LIN {X 0,Y 573.313,Z 246.817,A -85,B 0,C 180,E1 -2273.642,E2 -2273.642} C_VEL
LIN {X 0,Y 573.236,Z 246.702,A -85,B 0,C 180,E1 -2276.492,E2 -2276.492} C_VEL
LIN {X 0,Y 573.238,Z 246.706,A -85,B 0,C 180,E1 -2278.564,E2 -2278.564} C_VEL
LIN {X 0,Y 573.228,Z 246.705,A -85,B 0,C 180,E1 -2280.992,E2 -2280.992} C_VEL
LIN {X 0,Y 573.26,Z 246.695,A -85,B 0,C 180,E1 -2283.523,E2 -2283.523} C_VEL
LIN {X 0,Y 573.212,Z 246.707,A -85,B 0,C 180,E1 -2286.051,E2 -2286.051} C_VEL
LIN {X 0,Y 573.239,Z 246.706,A -85,B 0,C 180,E1 -2288.701,E2 -2288.701} C_VEL
LIN {X 0,Y 573.25,Z 246.695,A -85,B 0,C 180,E1 -2291.595,E2 -2291.595} C_VEL
LIN {X 0,Y 573.235,Z 246.71,A -85,B 0,C 180,E1 -2294.332,E2 -2294.332} C_VEL
LIN {X 0,Y 573.235,Z 246.7,A -85,B 0,C 180,E1 -2297.358,E2 -2297.358} C_VEL
LIN {X 0,Y 573.244,Z 246.706,A -85,B 0,C 180,E1 -2300.393,E2 -2300.393} C_VEL
LIN {X 0,Y 573.251,Z 246.697,A -85,B 0,C 180,E1 -2303.077,E2 -2303.077} C_VEL
LIN {X 0,Y 573.268,Z 246.693,A -85,B 0,C 180,E1 -2305.671,E2 -2305.671} C_VEL
LIN {X 0,Y 573.242,Z 246.707,A -85,B 0,C 180,E1 -2308.185,E2 -2308.185} C_VEL
LIN {X 0,Y 573.262,Z 246.698,A -85,B 0,C 180,E1 -2310.634,E2 -2310.634} C_VEL
LIN {X 0,Y 573.264,Z 246.698,A -85,B 0,C 180,E1 -2313.5,E2 -2313.5} C_VEL
LIN {X 0,Y 573.227,Z 246.707,A -85,B 0,C 180,E1 -2316.134,E2 -2316.134} C_VEL
LIN {X 0,Y 573.243,Z 246.699,A -85,B 0,C 180,E1 -2319.173,E2 -2319.173} C_VEL
LIN {X 0,Y 573.23,Z 246.704,A -85,B 0,C 180,E1 -2321.412,E2 -2321.412} C_VEL
LIN {X 0,Y 573.252,Z 246.703,A -85,B 0,C 180,E1 -2323.622,E2 -2323.622} C_VEL
LIN {X 0,Y 573.231,Z 246.701,A -85,B 0,C 180,E1 -2326.529,E2 -2326.529} C_VEL
LIN {X 0,Y 573.253,Z 246.696,A -85,B 0,C 180,E1 -2328.745,E2 -2328.745} C_VEL
LIN {X 0,Y 573.283,Z 246.701,A -85,B 0,C 180,E1 -2331.541,E2 -2331.541} C_VEL
LIN {X 0,Y 573.286,Z 246.693,A -85,B 0,C 180,E1 -2334.372,E2 -2334.372} C_VEL
LIN {X 0,Y 573.301,Z 246.696,A -85,B 0,C 180,E1 -2337.892,E2 -2337.892} C_VEL
LIN {X 0,Y 573.328,Z 246.688,A -85,B 0,C 180,E1 -2340.702,E2 -2340.702} C_VEL
LIN {X 0,Y 573.233,Z 246.709,A -85,B 0,C 180,E1 -2343.515,E2 -2343.515} C_VEL
LIN {X 0,Y 573.286,Z 246.7,A -85,B 0,C 180,E1 -2345.628,E2 -2345.628} C_VEL
LIN {X 0,Y 573.283,Z 246.692,A -85,B 0,C 180,E1 -2348.46,E2 -2348.46} C_VEL
LIN {X 0,Y 573.262,Z 246.706,A -85,B 0,C 180,E1 -2351.312,E2 -2351.312} C_VEL
LIN {X 0,Y 573.265,Z 246.695,A -85,B 0,C 180,E1 -2354.193,E2 -2354.193} C_VEL
LIN {X 0,Y 573.252,Z 246.706,A -85,B 0,C 180,E1 -2357.112,E2 -2357.112} C_VEL
LIN {X 0,Y 573.247,Z 246.697,A -85,B 0,C 180,E1 -2360.077,E2 -2360.077} C_VEL
LIN {X 0,Y 573.226,Z 246.711,A -85,B 0,C 180,E1 -2363.1,E2 -2363.1} C_VEL
LIN {X 0,Y 573.244,Z 246.7,A -85,B 0,C 180,E1 -2364.396,E2 -2364.396} C_VEL
LIN {X 0,Y 572.617,Z 246.786,A -85,B 0,C 180,E1 -2364.983,E2 -2364.983} C_VEL
LIN {X 0,Y 569.776,Z 247.14,A -85,B 0,C 180,E1 -2365.934,E2 -2365.934} C_VEL
LIN {X 0,Y 567.346,Z 247.442,A -85,B 0,C 180,E1 -2366.7,E2 -2366.7} C_VEL
LIN {X 0,Y 566.295,Z 247.57,A -85,B 0,C 180,E1 -2367.291,E2 -2367.291} C_VEL
LIN {X 0,Y 566.207,Z 247.578,A -85,B 0,C 180,E1 -2367.491,E2 -2367.491} C_VEL
LIN {X 0,Y 566.22,Z 247.574,A -85,B 0,C 180,E1 -2369.768,E2 -2369.768} C_VEL
LIN {X 0,Y 566.201,Z 247.575,A -85,B 0,C 180,E1 -2372.431,E2 -2372.431} C_VEL
LIN {X 0,Y 566.209,Z 247.582,A -85,B 0,C 180,E1 -2374.995,E2 -2374.995} C_VEL
LIN {X 0,Y 566.192,Z 247.579,A -85,B 0,C 180,E1 -2377.461,E2 -2377.461} C_VEL
LIN {X 0,Y 566.222,Z 247.574,A -85,B 0,C 180,E1 -2380.198,E2 -2380.198} C_VEL
LIN {X 0,Y 566.197,Z 247.581,A -85,B 0,C 180,E1 -2383.055,E2 -2383.055} C_VEL
LIN {X 0,Y 566.199,Z 247.578,A -85,B 0,C 180,E1 -2386.049,E2 -2386.049} C_VEL
LIN {X 0,Y 566.209,Z 247.581,A -85,B 0,C 180,E1 -2388.865,E2 -2388.865} C_VEL
LIN {X 0,Y 566.184,Z 247.577,A -85,B 0,C 180,E1 -2391.638,E2 -2391.638} C_VEL
LIN {X 0,Y 566.195,Z 247.584,A -85,B 0,C 180,E1 -2394.311,E2 -2394.311} C_VEL
LIN {X 0,Y 566.228,Z 247.577,A -85,B 0,C 180,E1 -2396.899,E2 -2396.899} C_VEL
LIN {X 0,Y 566.18,Z 247.58,A -85,B 0,C 180,E1 -2399.408,E2 -2399.408} C_VEL
LIN {X 0,Y 566.212,Z 247.575,A -85,B 0,C 180,E1 -2401.858,E2 -2401.858} C_VEL
LIN {X 0,Y 566.216,Z 247.582,A -85,B 0,C 180,E1 -2404.252,E2 -2404.252} C_VEL
LIN {X 0,Y 566.24,Z 247.699,A -85,B 0,C 180,E1 -2407.28,E2 -2407.28} C_VEL
LIN {X 0,Y 567.062,Z 253.165,A -85,B 0,C 180,E1 -2408.173,E2 -2408.173} C_VEL
LIN {X 0,Y 566.746,Z 272.236,A -85,B 0,C 180,E1 -2411.01,E2 -2411.01} C_VEL
LIN {X 0,Y 566.631,Z 286.377,A -85,B 0,C 180,E1 -2413.053,E2 -2413.053} C_VEL
LIN {X 0,Y 567.533,Z 291.478,A -85,B 0,C 180,E1 -2413.174,E2 -2413.174} C_VEL
LIN {X 0,Y 567.785,Z 300.796,A -85,B 0,C 180,E1 -2413.302,E2 -2413.302} C_VEL
LIN {X 0,Y 567.442,Z 423.944,A -85,B 0,C 180,E1 -2414.902,E2 -2414.902} C_VEL
LIN {X 0,Y 567.321,Z 438.302,A -85,B 0,C 180,E1 -2415.239,E2 -2415.239} C_VEL
LIN {X 0,Y 567.131,Z 452.855,A -85,B 0,C 180,E1 -2415.742,E2 -2415.742} C_VEL
LIN {X 0,Y 566.944,Z 466.542,A -85,B 0,C 180,E1 -2416.377,E2 -2416.377} C_VEL
LIN {X 0,Y 566.744,Z 478.824,A -85,B 0,C 180,E1 -2417.103,E2 -2417.103} C_VEL
LIN {X 0,Y 566.56,Z 491.218,A -85,B 0,C 180,E1 -2418.008,E2 -2418.008} C_VEL
LIN {X 0,Y 566.434,Z 502.054,A -85,B 0,C 180,E1 -2418.98,E2 -2418.98} C_VEL
LIN {X 0,Y 566.215,Z 511.482,A -85,B 0,C 180,E1 -2419.993,E2 -2419.993} C_VEL
LIN {X 0,Y 566.133,Z 519.865,A -85,B 0,C 180,E1 -2421.073,E2 -2421.073} C_VEL
LIN {X 0,Y 566.047,Z 527.875,A -85,B 0,C 180,E1 -2422.33,E2 -2422.33} C_VEL
LIN {X 0,Y 565.945,Z 534.324,A -85,B 0,C 180,E1 -2423.583,E2 -2423.583} C_VEL
LIN {X 0,Y 565.928,Z 538.8,A -85,B 0,C 180,E1 -2424.656,E2 -2424.656} C_VEL
LIN {X 0,Y 565.957,Z 542.312,A -85,B 0,C 180,E1 -2425.727,E2 -2425.727} C_VEL
LIN {X 0,Y 565.875,Z 545.744,A -85,B 0,C 180,E1 -2427.152,E2 -2427.152} C_VEL
LIN {X 0,Y 565.844,Z 547.785,A -85,B 0,C 180,E1 -2428.577,E2 -2428.577} C_VEL
LIN {X 0,Y 565.838,Z 548.496,A -85,B 0,C 180,E1 -2430,E2 -2430} C_VEL
LIN {X 0,Y 565.841,Z 547.88,A -85,B 0,C 180,E1 -2431.423,E2 -2431.423} C_VEL
LIN {X 0,Y 565.873,Z 545.923,A -85,B 0,C 180,E1 -2432.847,E2 -2432.847} C_VEL
LIN {X 0,Y 565.958,Z 542.577,A -85,B 0,C 180,E1 -2434.273,E2 -2434.273} C_VEL
LIN {X 0,Y 565.983,Z 537.749,A -85,B 0,C 180,E1 -2435.701,E2 -2435.701} C_VEL
LIN {X 0,Y 565.981,Z 531.282,A -85,B 0,C 180,E1 -2437.133,E2 -2437.133} C_VEL
LIN {X 0,Y 566.093,Z 524.083,A -85,B 0,C 180,E1 -2438.388,E2 -2438.388} C_VEL
LIN {X 0,Y 566.172,Z 516.544,A -85,B 0,C 180,E1 -2439.466,E2 -2439.466} C_VEL
LIN {X 0,Y 566.29,Z 507.487,A -85,B 0,C 180,E1 -2440.548,E2 -2440.548} C_VEL
LIN {X 0,Y 566.47,Z 496.523,A -85,B 0,C 180,E1 -2441.631,E2 -2441.631} C_VEL
LIN {X 0,Y 566.631,Z 485.35,A -85,B 0,C 180,E1 -2442.536,E2 -2442.536} C_VEL
LIN {X 0,Y 566.843,Z 473,A -85,B 0,C 180,E1 -2443.351,E2 -2443.351} C_VEL
LIN {X 0,Y 567.064,Z 461.118,A -85,B 0,C 180,E1 -2443.985,E2 -2443.985} C_VEL
LIN {X 0,Y 567.234,Z 448.803,A -85,B 0,C 180,E1 -2444.507,E2 -2444.507} C_VEL
LIN {X 0,Y 567.352,Z 434.83,A -85,B 0,C 180,E1 -2444.947,E2 -2444.947} C_VEL
LIN {X 0,Y 567.451,Z 421.093,A -85,B 0,C 180,E1 -2445.236,E2 -2445.236} C_VEL
LIN {X 0,Y 567.731,Z 292.506,A -85,B 0,C 180,E1 -2446.897,E2 -2446.897} C_VEL
LIN {X 0,Y 566.636,Z 286.481,A -85,B 0,C 180,E1 -2447.029,E2 -2447.029} C_VEL
LIN {X 0,Y 566.788,Z 269.863,A -85,B 0,C 180,E1 -2449.429,E2 -2449.429} C_VEL
LIN {X 0,Y 567.066,Z 252.496,A -85,B 0,C 180,E1 -2452.018,E2 -2452.018} C_VEL
LIN {X 0,Y 566.246,Z 247.694,A -85,B 0,C 180,E1 -2452.812,E2 -2452.812} C_VEL
LIN {X 0,Y 566.215,Z 247.58,A -85,B 0,C 180,E1 -2455.748,E2 -2455.748} C_VEL
LIN {X 0,Y 566.202,Z 247.576,A -85,B 0,C 180,E1 -2458.201,E2 -2458.201} C_VEL
LIN {X 0,Y 566.189,Z 247.58,A -85,B 0,C 180,E1 -2461.076,E2 -2461.076} C_VEL
LIN {X 0,Y 566.21,Z 247.582,A -85,B 0,C 180,E1 -2463.733,E2 -2463.733} C_VEL
LIN {X 0,Y 566.208,Z 247.576,A -85,B 0,C 180,E1 -2466.568,E2 -2466.568} C_VEL
LIN {X 0,Y 566.207,Z 247.583,A -85,B 0,C 180,E1 -2469.684,E2 -2469.684} C_VEL
LIN {X 0,Y 566.211,Z 247.573,A -85,B 0,C 180,E1 -2472.086,E2 -2472.086} C_VEL
LIN {X 0,Y 566.169,Z 247.584,A -85,B 0,C 180,E1 -2475.035,E2 -2475.035} C_VEL
LIN {X 0,Y 566.207,Z 247.571,A -85,B 0,C 180,E1 -2478.136,E2 -2478.136} C_VEL
LIN {X 0,Y 566.217,Z 247.575,A -85,B 0,C 180,E1 -2480.726,E2 -2480.726} C_VEL
LIN {X 0,Y 566.212,Z 247.576,A -85,B 0,C 180,E1 -2483.783,E2 -2483.783} C_VEL
LIN {X 0,Y 566.206,Z 247.57,A -85,B 0,C 180,E1 -2486.265,E2 -2486.265} C_VEL
LIN {X 0,Y 566.196,Z 247.58,A -85,B 0,C 180,E1 -2488.921,E2 -2488.921} C_VEL
LIN {X 0,Y 566.189,Z 247.587,A -85,B 0,C 180,E1 -2491.046,E2 -2491.046} C_VEL
LIN {X 0,Y 566.208,Z 247.577,A -85,B 0,C 180,E1 -2493.458,E2 -2493.458} C_VEL
LIN {X 0,Y 566.192,Z 247.578,A -85,B 0,C 180,E1 -2495.819,E2 -2495.819} C_VEL
LIN {X 0,Y 566.2,Z 247.584,A -85,B 0,C 180,E1 -2498.902,E2 -2498.902} C_VEL
LIN {X 0,Y 566.204,Z 247.581,A -85,B 0,C 180,E1 -2501.172,E2 -2501.172} C_VEL
LIN {X 0,Y 566.213,Z 247.576,A -85,B 0,C 180,E1 -2503.412,E2 -2503.412} C_VEL
LIN {X 0,Y 566.194,Z 247.578,A -85,B 0,C 180,E1 -2506.359,E2 -2506.359} C_VEL
LIN {X 0,Y 566.266,Z 247.576,A -85,B 0,C 180,E1 -2508.654,E2 -2508.654} C_VEL
LIN {X 0,Y 566.226,Z 247.571,A -85,B 0,C 180,E1 -2511.434,E2 -2511.434} C_VEL
LIN {X 0,Y 566.254,Z 247.574,A -85,B 0,C 180,E1 -2514.302,E2 -2514.302} C_VEL
LIN {X 0,Y 566.271,Z 247.565,A -85,B 0,C 180,E1 -2517.866,E2 -2517.866} C_VEL
LIN {X 0,Y 566.299,Z 247.571,A -85,B 0,C 180,E1 -2520.711,E2 -2520.711} C_VEL
LIN {X 0,Y 566.27,Z 247.569,A -85,B 0,C 180,E1 -2522.846,E2 -2522.846} C_VEL
LIN {X 0,Y 566.253,Z 247.569,A -85,B 0,C 180,E1 -2525.698,E2 -2525.698} C_VEL
LIN {X 0,Y 566.24,Z 247.577,A -85,B 0,C 180,E1 -2528.565,E2 -2528.565} C_VEL
LIN {X 0,Y 566.232,Z 247.571,A -85,B 0,C 180,E1 -2531.454,E2 -2531.454} C_VEL
LIN {X 0,Y 566.225,Z 247.578,A -85,B 0,C 180,E1 -2534.507,E2 -2534.507} C_VEL
LIN {X 0,Y 566.195,Z 247.575,A -85,B 0,C 180,E1 -2537.332,E2 -2537.332} C_VEL
LIN {X 0,Y 566.206,Z 247.581,A -85,B 0,C 180,E1 -2540.337,E2 -2540.337} C_VEL
LIN {X 0,Y 566.182,Z 247.578,A -85,B 0,C 180,E1 -2543.404,E2 -2543.404} C_VEL
LIN {X 0,Y 566.207,Z 247.581,A -85,B 0,C 180,E1 -2545.749,E2 -2545.749} C_VEL
LIN {X 0,Y 566.198,Z 247.583,A -85,B 0,C 180,E1 -2548.203,E2 -2548.203} C_VEL
LIN {X 0,Y 566.186,Z 247.579,A -85,B 0,C 180,E1 -2550.592,E2 -2550.592} C_VEL
LIN {X 0,Y 566.221,Z 247.57,A -85,B 0,C 180,E1 -2553.102,E2 -2553.102} C_VEL
LIN {X 0,Y 566.206,Z 247.576,A -85,B 0,C 180,E1 -2555.689,E2 -2555.689} C_VEL
LIN {X 0,Y 566.21,Z 247.576,A -85,B 0,C 180,E1 -2558.56,E2 -2558.56} C_VEL
LIN {X 0,Y 566.206,Z 247.576,A -85,B 0,C 180,E1 -2561.137,E2 -2561.137} C_VEL
LIN {X 0,Y 566.192,Z 247.582,A -85,B 0,C 180,E1 -2564.036,E2 -2564.036} C_VEL
LIN {X 0,Y 566.205,Z 247.577,A -85,B 0,C 180,E1 -2567.083,E2 -2567.083} C_VEL
LIN {X 0,Y 566.223,Z 247.58,A -85,B 0,C 180,E1 -2569.803,E2 -2569.803} C_VEL
LIN {X 0,Y 566.195,Z 247.575,A -85,B 0,C 180,E1 -2572.6,E2 -2572.6} C_VEL
LIN {X 0,Y 566.201,Z 247.582,A -85,B 0,C 180,E1 -2575.183,E2 -2575.183} C_VEL
LIN {X 0,Y 566.233,Z 247.578,A -85,B 0,C 180,E1 -2577.744,E2 -2577.744} C_VEL
LIN {X 0,Y 566.202,Z 247.57,A -85,B 0,C 180,E1 -2580.329,E2 -2580.329} C_VEL
LIN {X 0,Y 566.21,Z 247.578,A -85,B 0,C 180,E1 -2582.662,E2 -2582.662} C_VEL
LIN {X 0,Y 566.236,Z 247.578,A -85,B 0,C 180,E1 -2585.04,E2 -2585.04} C_VEL
LIN {X 0,Y 566.263,Z 247.807,A -85,B 0,C 180,E1 -2586.212,E2 -2586.212} C_VEL
LIN {X 0,Y 567.195,Z 253.103,A -85,B 0,C 180,E1 -2587.027,E2 -2587.027} C_VEL
LIN {X 0,Y 566.934,Z 273.326,A -85,B 0,C 180,E1 -2589.88,E2 -2589.88} C_VEL
LIN {X 0,Y 566.604,Z 294.059,A -85,B 0,C 180,E1 -2592.763,E2 -2592.763} C_VEL
LIN {X 0,Y 566.662,Z 296.302,A -85,B 0,C 180,E1 -2593.024,E2 -2593.024} C_VEL
LIN {X 0,Y 567.795,Z 303.619,A -85,B 0,C 180,E1 -2593.165,E2 -2593.165} C_VEL
LIN {X 0,Y 567.456,Z 432.658,A -85,B 0,C 180,E1 -2594.833,E2 -2594.833} C_VEL
LIN {X 0,Y 567.301,Z 447.176,A -85,B 0,C 180,E1 -2595.16,E2 -2595.16} C_VEL
LIN {X 0,Y 567.19,Z 460.406,A -85,B 0,C 180,E1 -2595.599,E2 -2595.599} C_VEL
LIN {X 0,Y 567.011,Z 473.883,A -85,B 0,C 180,E1 -2596.196,E2 -2596.196} C_VEL
LIN {X 0,Y 566.77,Z 486.683,A -85,B 0,C 180,E1 -2596.921,E2 -2596.921} C_VEL
LIN {X 0,Y 566.615,Z 498.316,A -85,B 0,C 180,E1 -2597.737,E2 -2597.737} C_VEL
LIN {X 0,Y 566.443,Z 508.224,A -85,B 0,C 180,E1 -2598.572,E2 -2598.572} C_VEL
LIN {X 0,Y 566.294,Z 518.709,A -85,B 0,C 180,E1 -2599.633,E2 -2599.633} C_VEL
LIN {X 0,Y 566.18,Z 527.56,A -85,B 0,C 180,E1 -2600.714,E2 -2600.714} C_VEL
LIN {X 0,Y 566.047,Z 536.037,A -85,B 0,C 180,E1 -2601.971,E2 -2601.971} C_VEL
LIN {X 0,Y 565.966,Z 543.803,A -85,B 0,C 180,E1 -2603.422,E2 -2603.422} C_VEL
LIN {X 0,Y 565.928,Z 548.961,A -85,B 0,C 180,E1 -2604.656,E2 -2604.656} C_VEL
LIN {X 0,Y 565.956,Z 552.444,A -85,B 0,C 180,E1 -2605.727,E2 -2605.727} C_VEL
LIN {X 0,Y 565.875,Z 555.832,A -85,B 0,C 180,E1 -2607.153,E2 -2607.153} C_VEL
LIN {X 0,Y 565.841,Z 557.833,A -85,B 0,C 180,E1 -2608.577,E2 -2608.577} C_VEL
LIN {X 0,Y 565.837,Z 558.5,A -85,B 0,C 180,E1 -2610,E2 -2610} C_VEL
LIN {X 0,Y 565.841,Z 557.834,A -85,B 0,C 180,E1 -2611.423,E2 -2611.423} C_VEL
LIN {X 0,Y 565.875,Z 555.834,A -85,B 0,C 180,E1 -2612.848,E2 -2612.848} C_VEL
LIN {X 0,Y 565.956,Z 552.446,A -85,B 0,C 180,E1 -2614.273,E2 -2614.273} C_VEL
LIN {X 0,Y 565.985,Z 547.568,A -85,B 0,C 180,E1 -2615.701,E2 -2615.701} C_VEL
LIN {X 0,Y 565.995,Z 543.044,A -85,B 0,C 180,E1 -2616.739,E2 -2616.739} C_VEL
LIN {X 0,Y 566.047,Z 536.037,A -85,B 0,C 180,E1 -2618.029,E2 -2618.029} C_VEL
LIN {X 0,Y 566.177,Z 527.559,A -85,B 0,C 180,E1 -2619.286,E2 -2619.286} C_VEL
LIN {X 0,Y 566.294,Z 518.708,A -85,B 0,C 180,E1 -2620.367,E2 -2620.367} C_VEL
LIN {X 0,Y 566.485,Z 507.991,A -85,B 0,C 180,E1 -2621.449,E2 -2621.449} C_VEL
LIN {X 0,Y 566.611,Z 497.141,A -85,B 0,C 180,E1 -2622.354,E2 -2622.354} C_VEL
LIN {X 0,Y 566.778,Z 485.258,A -85,B 0,C 180,E1 -2623.17,E2 -2623.17} C_VEL
LIN {X 0,Y 567.033,Z 472.101,A -85,B 0,C 180,E1 -2623.895,E2 -2623.895} C_VEL
LIN {X 0,Y 567.21,Z 459.022,A -85,B 0,C 180,E1 -2624.454,E2 -2624.454} C_VEL
LIN {X 0,Y 567.359,Z 445.048,A -85,B 0,C 180,E1 -2624.896,E2 -2624.896} C_VEL
LIN {X 0,Y 567.464,Z 431.148,A -85,B 0,C 180,E1 -2625.19,E2 -2625.19} C_VEL
LIN {X 0,Y 567.74,Z 302.087,A -85,B 0,C 180,E1 -2626.857,E2 -2626.857} C_VEL
LIN {X 0,Y 566.649,Z 296.08,A -85,B 0,C 180,E1 -2626.989,E2 -2626.989} C_VEL
LIN {X 0,Y 566.833,Z 277.357,A -85,B 0,C 180,E1 -2629.558,E2 -2629.558} C_VEL
LIN {X 0,Y 567.175,Z 258.498,A -85,B 0,C 180,E1 -2632.205,E2 -2632.205} C_VEL
LIN {X 0,Y 567.054,Z 251.755,A -85,B 0,C 180,E1 -2633.172,E2 -2633.172} C_VEL
LIN {X 0,Y 566.249,Z 247.675,A -85,B 0,C 180,E1 -2633.837,E2 -2633.837} C_VEL
LIN {X 0,Y 566.208,Z 247.579,A -85,B 0,C 180,E1 -2636.659,E2 -2636.659} C_VEL
LIN {X 0,Y 566.191,Z 247.576,A -85,B 0,C 180,E1 -2638.953,E2 -2638.953} C_VEL
LIN {X 0,Y 566.195,Z 247.578,A -85,B 0,C 180,E1 -2641.421,E2 -2641.421} C_VEL
LIN {X 0,Y 566.208,Z 247.576,A -85,B 0,C 180,E1 -2643.955,E2 -2643.955} C_VEL
LIN {X 0,Y 566.197,Z 247.583,A -85,B 0,C 180,E1 -2646.569,E2 -2646.569} C_VEL
LIN {X 0,Y 566.212,Z 247.576,A -85,B 0,C 180,E1 -2649.685,E2 -2649.685} C_VEL
LIN {X 0,Y 566.211,Z 247.577,A -85,B 0,C 180,E1 -2652.087,E2 -2652.087} C_VEL
LIN {X 0,Y 566.169,Z 247.581,A -85,B 0,C 180,E1 -2655.035,E2 -2655.035} C_VEL
LIN {X 0,Y 566.209,Z 247.583,A -85,B 0,C 180,E1 -2658.136,E2 -2658.136} C_VEL
LIN {X 0,Y 566.218,Z 247.577,A -85,B 0,C 180,E1 -2660.727,E2 -2660.727} C_VEL
LIN {X 0,Y 566.212,Z 247.577,A -85,B 0,C 180,E1 -2663.783,E2 -2663.783} C_VEL
LIN {X 0,Y 566.206,Z 247.58,A -85,B 0,C 180,E1 -2666.265,E2 -2666.265} C_VEL
LIN {X 0,Y 566.196,Z 247.577,A -85,B 0,C 180,E1 -2668.921,E2 -2668.921} C_VEL
LIN {X 0,Y 566.188,Z 247.577,A -85,B 0,C 180,E1 -2671.046,E2 -2671.046} C_VEL
LIN {X 0,Y 566.239,Z 247.572,A -85,B 0,C 180,E1 -2673.46,E2 -2673.46} C_VEL
LIN {X 0,Y 566.193,Z 247.585,A -85,B 0,C 180,E1 -2675.819,E2 -2675.819} C_VEL
LIN {X 0,Y 566.2,Z 247.575,A -85,B 0,C 180,E1 -2678.902,E2 -2678.902} C_VEL
LIN {X 0,Y 566.204,Z 247.577,A -85,B 0,C 180,E1 -2681.172,E2 -2681.172} C_VEL
LIN {X 0,Y 566.213,Z 247.577,A -85,B 0,C 180,E1 -2683.412,E2 -2683.412} C_VEL
LIN {X 0,Y 566.194,Z 247.579,A -85,B 0,C 180,E1 -2686.359,E2 -2686.359} C_VEL
LIN {X 0,Y 566.225,Z 247.572,A -85,B 0,C 180,E1 -2688.675,E2 -2688.675} C_VEL
LIN {X 0,Y 566.227,Z 247.578,A -85,B 0,C 180,E1 -2691.434,E2 -2691.434} C_VEL
LIN {X 0,Y 566.254,Z 247.569,A -85,B 0,C 180,E1 -2694.302,E2 -2694.302} C_VEL
LIN {X 0,Y 566.272,Z 247.572,A -85,B 0,C 180,E1 -2697.866,E2 -2697.866} C_VEL
LIN {X 0,Y 566.297,Z 247.564,A -85,B 0,C 180,E1 -2700.711,E2 -2700.711} C_VEL
LIN {X 0,Y 566.27,Z 247.566,A -85,B 0,C 180,E1 -2702.846,E2 -2702.846} C_VEL
LIN {X 0,Y 566.254,Z 247.575,A -85,B 0,C 180,E1 -2705.698,E2 -2705.698} C_VEL
LIN {X 0,Y 566.227,Z 247.571,A -85,B 0,C 180,E1 -2708.566,E2 -2708.566} C_VEL
LIN {X 0,Y 566.233,Z 247.579,A -85,B 0,C 180,E1 -2711.455,E2 -2711.455} C_VEL
LIN {X 0,Y 566.226,Z 247.572,A -85,B 0,C 180,E1 -2714.507,E2 -2714.507} C_VEL
LIN {X 0,Y 566.196,Z 247.584,A -85,B 0,C 180,E1 -2717.332,E2 -2717.332} C_VEL
LIN {X 0,Y 566.207,Z 247.574,A -85,B 0,C 180,E1 -2720.338,E2 -2720.338} C_VEL
LIN {X 0,Y 566.182,Z 247.583,A -85,B 0,C 180,E1 -2723.404,E2 -2723.404} C_VEL
LIN {X 0,Y 566.208,Z 247.574,A -85,B 0,C 180,E1 -2725.749,E2 -2725.749} C_VEL
LIN {X 0,Y 566.207,Z 247.578,A -85,B 0,C 180,E1 -2727.491,E2 -2727.491} C_VEL
LIN {X 0,Y 565.531,Z 247.661,A -85,B 0,C 180,E1 -2728.085,E2 -2728.085} C_VEL
LIN {X 0,Y 562.668,Z 248.025,A -85,B 0,C 180,E1 -2729.049,E2 -2729.049} C_VEL
LIN {X 0,Y 560.257,Z 248.32,A -85,B 0,C 180,E1 -2729.824,E2 -2729.824} C_VEL
LIN {X 0,Y 559.227,Z 248.447,A -85,B 0,C 180,E1 -2730.423,E2 -2730.423} C_VEL
LIN {X 0,Y 559.147,Z 248.456,A -85,B 0,C 180,E1 -2730.626,E2 -2730.626} C_VEL
LIN {X 0,Y 559.159,Z 248.447,A -85,B 0,C 180,E1 -2733.575,E2 -2733.575} C_VEL
LIN {X 0,Y 559.164,Z 248.455,A -85,B 0,C 180,E1 -2736.449,E2 -2736.449} C_VEL
LIN {X 0,Y 559.174,Z 248.457,A -85,B 0,C 180,E1 -2738.934,E2 -2738.934} C_VEL
LIN {X 0,Y 559.182,Z 248.444,A -85,B 0,C 180,E1 -2741.769,E2 -2741.769} C_VEL
LIN {X 0,Y 559.136,Z 248.466,A -85,B 0,C 180,E1 -2744.74,E2 -2744.74} C_VEL
LIN {X 0,Y 559.161,Z 248.45,A -85,B 0,C 180,E1 -2747.258,E2 -2747.258} C_VEL
LIN {X 0,Y 559.182,Z 248.454,A -85,B 0,C 180,E1 -2750.136,E2 -2750.136} C_VEL
LIN {X 0,Y 559.143,Z 248.46,A -85,B 0,C 180,E1 -2752.893,E2 -2752.893} C_VEL
LIN {X 0,Y 559.165,Z 248.455,A -85,B 0,C 180,E1 -2756.051,E2 -2756.051} C_VEL
LIN {X 0,Y 559.155,Z 248.457,A -85,B 0,C 180,E1 -2758.981,E2 -2758.981} C_VEL
LIN {X 0,Y 559.168,Z 248.45,A -85,B 0,C 180,E1 -2761.619,E2 -2761.619} C_VEL
LIN {X 0,Y 559.183,Z 248.456,A -85,B 0,C 180,E1 -2763.904,E2 -2763.904} C_VEL
LIN {X 0,Y 559.183,Z 248.549,A -85,B 0,C 180,E1 -2767.094,E2 -2767.094} C_VEL
LIN {X 0,Y 560.091,Z 253.226,A -85,B 0,C 180,E1 -2767.887,E2 -2767.887} C_VEL
LIN {X 0,Y 559.879,Z 269.152,A -85,B 0,C 180,E1 -2770.298,E2 -2770.298} C_VEL
LIN {X 0,Y 559.65,Z 286.418,A -85,B 0,C 180,E1 -2772.837,E2 -2772.837} C_VEL
LIN {X 0,Y 560.963,Z 293.554,A -85,B 0,C 180,E1 -2772.997,E2 -2772.997} C_VEL
LIN {X 0,Y 560.62,Z 422.744,A -85,B 0,C 180,E1 -2774.69,E2 -2774.69} C_VEL
LIN {X 0,Y 560.429,Z 436.966,A -85,B 0,C 180,E1 -2775.012,E2 -2775.012} C_VEL
LIN {X 0,Y 560.27,Z 450.607,A -85,B 0,C 180,E1 -2775.471,E2 -2775.471} C_VEL
LIN {X 0,Y 560.089,Z 463.019,A -85,B 0,C 180,E1 -2776.022,E2 -2776.022} C_VEL
LIN {X 0,Y 559.854,Z 475.987,A -85,B 0,C 180,E1 -2776.756,E2 -2776.756} C_VEL
LIN {X 0,Y 559.646,Z 487.738,A -85,B 0,C 180,E1 -2777.582,E2 -2777.582} C_VEL
LIN {X 0,Y 559.472,Z 498.218,A -85,B 0,C 180,E1 -2778.472,E2 -2778.472} C_VEL
LIN {X 0,Y 559.312,Z 508.308,A -85,B 0,C 180,E1 -2779.502,E2 -2779.502} C_VEL
LIN {X 0,Y 559.123,Z 517.224,A -85,B 0,C 180,E1 -2780.596,E2 -2780.596} C_VEL
LIN {X 0,Y 558.987,Z 525.761,A -85,B 0,C 180,E1 -2781.869,E2 -2781.869} C_VEL
LIN {X 0,Y 558.903,Z 532.641,A -85,B 0,C 180,E1 -2783.14,E2 -2783.14} C_VEL
LIN {X 0,Y 558.914,Z 537.391,A -85,B 0,C 180,E1 -2784.227,E2 -2784.227} C_VEL
LIN {X 0,Y 558.866,Z 542.315,A -85,B 0,C 180,E1 -2785.673,E2 -2785.673} C_VEL
LIN {X 0,Y 558.796,Z 545.745,A -85,B 0,C 180,E1 -2787.116,E2 -2787.116} C_VEL
LIN {X 0,Y 558.744,Z 547.786,A -85,B 0,C 180,E1 -2788.558,E2 -2788.558} C_VEL
LIN {X 0,Y 558.739,Z 548.496,A -85,B 0,C 180,E1 -2790,E2 -2790} C_VEL
LIN {X 0,Y 558.741,Z 547.879,A -85,B 0,C 180,E1 -2791.441,E2 -2791.441} C_VEL
LIN {X 0,Y 558.794,Z 545.922,A -85,B 0,C 180,E1 -2792.884,E2 -2792.884} C_VEL
LIN {X 0,Y 558.867,Z 542.576,A -85,B 0,C 180,E1 -2794.327,E2 -2794.327} C_VEL
LIN {X 0,Y 558.912,Z 537.746,A -85,B 0,C 180,E1 -2795.773,E2 -2795.773} C_VEL
LIN {X 0,Y 558.907,Z 531.28,A -85,B 0,C 180,E1 -2797.224,E2 -2797.224} C_VEL
LIN {X 0,Y 559.028,Z 524.08,A -85,B 0,C 180,E1 -2798.495,E2 -2798.495} C_VEL
LIN {X 0,Y 559.124,Z 516.539,A -85,B 0,C 180,E1 -2799.587,E2 -2799.587} C_VEL
LIN {X 0,Y 559.287,Z 507.482,A -85,B 0,C 180,E1 -2800.681,E2 -2800.681} C_VEL
LIN {X 0,Y 559.482,Z 496.517,A -85,B 0,C 180,E1 -2801.778,E2 -2801.778} C_VEL
LIN {X 0,Y 559.687,Z 485.343,A -85,B 0,C 180,E1 -2802.694,E2 -2802.694} C_VEL
LIN {X 0,Y 559.921,Z 472.992,A -85,B 0,C 180,E1 -2803.519,E2 -2803.519} C_VEL
LIN {X 0,Y 560.155,Z 461.108,A -85,B 0,C 180,E1 -2804.161,E2 -2804.161} C_VEL
LIN {X 0,Y 560.365,Z 447.732,A -85,B 0,C 180,E1 -2804.726,E2 -2804.726} C_VEL
LIN {X 0,Y 560.492,Z 433.616,A -85,B 0,C 180,E1 -2805.164,E2 -2805.164} C_VEL
LIN {X 0,Y 560.59,Z 419.549,A -85,B 0,C 180,E1 -2805.45,E2 -2805.45} C_VEL
LIN {X 0,Y 560.93,Z 293.281,A -85,B 0,C 180,E1 -2807.097,E2 -2807.097} C_VEL
LIN {X 0,Y 559.663,Z 286.667,A -85,B 0,C 180,E1 -2807.238,E2 -2807.238} C_VEL
LIN {X 0,Y 559.657,Z 284.25,A -85,B 0,C 180,E1 -2807.54,E2 -2807.54} C_VEL
LIN {X 0,Y 559.912,Z 265.234,A -85,B 0,C 180,E1 -2810.384,E2 -2810.384} C_VEL
LIN {X 0,Y 560.145,Z 253.815,A -85,B 0,C 180,E1 -2812.11,E2 -2812.11} C_VEL
LIN {X 0,Y 559.173,Z 248.535,A -85,B 0,C 180,E1 -2813.003,E2 -2813.003} C_VEL
LIN {X 0,Y 559.182,Z 248.457,A -85,B 0,C 180,E1 -2816.096,E2 -2816.096} C_VEL
LIN {X 0,Y 559.163,Z 248.451,A -85,B 0,C 180,E1 -2818.529,E2 -2818.529} C_VEL
LIN {X 0,Y 559.145,Z 248.46,A -85,B 0,C 180,E1 -2821.273,E2 -2821.273} C_VEL
LIN {X 0,Y 559.164,Z 248.457,A -85,B 0,C 180,E1 -2823.948,E2 -2823.948} C_VEL
LIN {X 0,Y 559.142,Z 248.46,A -85,B 0,C 180,E1 -2827.107,E2 -2827.107} C_VEL
LIN {X 0,Y 559.16,Z 248.457,A -85,B 0,C 180,E1 -2829.941,E2 -2829.941} C_VEL
LIN {X 0,Y 559.16,Z 248.45,A -85,B 0,C 180,E1 -2832.742,E2 -2832.742} C_VEL
LIN {X 0,Y 559.148,Z 248.458,A -85,B 0,C 180,E1 -2835.76,E2 -2835.76} C_VEL
LIN {X 0,Y 559.181,Z 248.445,A -85,B 0,C 180,E1 -2838.231,E2 -2838.231} C_VEL
LIN {X 0,Y 559.173,Z 248.459,A -85,B 0,C 180,E1 -2841.19,E2 -2841.19} C_VEL
LIN {X 0,Y 559.167,Z 248.453,A -85,B 0,C 180,E1 -2843.791,E2 -2843.791} C_VEL
LIN {X 0,Y 559.158,Z 248.447,A -85,B 0,C 180,E1 -2846.425,E2 -2846.425} C_VEL
LIN {X 0,Y 559.16,Z 248.457,A -85,B 0,C 180,E1 -2848.981,E2 -2848.981} C_VEL
LIN {X 0,Y 559.163,Z 248.455,A -85,B 0,C 180,E1 -2851.618,E2 -2851.618} C_VEL
LIN {X 0,Y 559.173,Z 248.449,A -85,B 0,C 180,E1 -2853.902,E2 -2853.902} C_VEL
LIN {X 0,Y 559.149,Z 248.458,A -85,B 0,C 180,E1 -2856.567,E2 -2856.567} C_VEL
LIN {X 0,Y 559.172,Z 248.453,A -85,B 0,C 180,E1 -2859.395,E2 -2859.395} C_VEL
LIN {X 0,Y 559.146,Z 248.455,A -85,B 0,C 180,E1 -2861.686,E2 -2861.686} C_VEL
LIN {X 0,Y 559.164,Z 248.452,A -85,B 0,C 180,E1 -2863.948,E2 -2863.948} C_VEL
LIN {X 0,Y 559.167,Z 248.452,A -85,B 0,C 180,E1 -2866.184,E2 -2866.184} C_VEL
LIN {X 0,Y 559.201,Z 248.451,A -85,B 0,C 180,E1 -2869.134,E2 -2869.134} C_VEL
LIN {X 0,Y 559.198,Z 248.447,A -85,B 0,C 180,E1 -2872.053,E2 -2872.053} C_VEL
LIN {X 0,Y 559.25,Z 248.446,A -85,B 0,C 180,E1 -2874.953,E2 -2874.953} C_VEL
LIN {X 0,Y 559.243,Z 248.44,A -85,B 0,C 180,E1 -2877.839,E2 -2877.839} C_VEL
LIN {X 0,Y 559.268,Z 248.446,A -85,B 0,C 180,E1 -2880.72,E2 -2880.72} C_VEL
LIN {X 0,Y 559.236,Z 248.445,A -85,B 0,C 180,E1 -2882.881,E2 -2882.881} C_VEL
LIN {X 0,Y 559.222,Z 248.445,A -85,B 0,C 180,E1 -2885.77,E2 -2885.77} C_VEL
LIN {X 0,Y 559.194,Z 248.452,A -85,B 0,C 180,E1 -2888.674,E2 -2888.674} C_VEL
LIN {X 0,Y 559.195,Z 248.448,A -85,B 0,C 180,E1 -2891.601,E2 -2891.601} C_VEL
LIN {X 0,Y 559.19,Z 248.453,A -85,B 0,C 180,E1 -2894.596,E2 -2894.596} C_VEL
LIN {X 0,Y 559.155,Z 248.453,A -85,B 0,C 180,E1 -2897.557,E2 -2897.557} C_VEL
LIN {X 0,Y 559.164,Z 248.458,A -85,B 0,C 180,E1 -2899.838,E2 -2899.838} C_VEL
LIN {X 0,Y 559.133,Z 248.463,A -85,B 0,C 180,E1 -2902.153,E2 -2902.153} C_VEL
LIN {X 0,Y 559.17,Z 248.452,A -85,B 0,C 180,E1 -2905.188,E2 -2905.188} C_VEL
LIN {X 0,Y 559.185,Z 248.453,A -85,B 0,C 180,E1 -2907.712,E2 -2907.712} C_VEL
LIN {X 0,Y 559.161,Z 248.459,A -85,B 0,C 180,E1 -2910.182,E2 -2910.182} C_VEL
LIN {X 0,Y 559.168,Z 248.449,A -85,B 0,C 180,E1 -2912.714,E2 -2912.714} C_VEL
LIN {X 0,Y 559.152,Z 248.449,A -85,B 0,C 180,E1 -2915.322,E2 -2915.322} C_VEL
LIN {X 0,Y 559.129,Z 248.464,A -85,B 0,C 180,E1 -2918.018,E2 -2918.018} C_VEL
LIN {X 0,Y 559.171,Z 248.451,A -85,B 0,C 180,E1 -2920.811,E2 -2920.811} C_VEL
LIN {X 0,Y 559.154,Z 248.462,A -85,B 0,C 180,E1 -2923.733,E2 -2923.733} C_VEL
LIN {X 0,Y 559.167,Z 248.452,A -85,B 0,C 180,E1 -2926.801,E2 -2926.801} C_VEL
LIN {X 0,Y 559.173,Z 248.452,A -85,B 0,C 180,E1 -2929.19,E2 -2929.19} C_VEL
LIN {X 0,Y 559.131,Z 248.458,A -85,B 0,C 180,E1 -2931.983,E2 -2931.983} C_VEL
LIN {X 0,Y 559.131,Z 248.459,A -85,B 0,C 180,E1 -2934.787,E2 -2934.787} C_VEL
LIN {X 0,Y 559.173,Z 248.459,A -85,B 0,C 180,E1 -2937.362,E2 -2937.362} C_VEL
LIN {X 0,Y 559.148,Z 248.449,A -85,B 0,C 180,E1 -2940.143,E2 -2940.143} C_VEL
LIN {X 0,Y 559.169,Z 248.458,A -85,B 0,C 180,E1 -2943.098,E2 -2943.098} C_VEL
LIN {X 0,Y 559.198,Z 248.566,A -85,B 0,C 180,E1 -2945.991,E2 -2945.991} C_VEL
LIN {X 0,Y 560.3,Z 254.545,A -85,B 0,C 180,E1 -2946.945,E2 -2946.945} C_VEL
LIN {X 0,Y 559.995,Z 274.614,A -85,B 0,C 180,E1 -2949.811,E2 -2949.811} C_VEL
LIN {X 0,Y 559.673,Z 295.923,A -85,B 0,C 180,E1 -2952.782,E2 -2952.782} C_VEL
LIN {X 0,Y 560.274,Z 299.54,A -85,B 0,C 180,E1 -2952.878,E2 -2952.878} C_VEL
LIN {X 0,Y 561.01,Z 304.395,A -85,B 0,C 180,E1 -2952.965,E2 -2952.965} C_VEL
LIN {X 0,Y 560.614,Z 432.657,A -85,B 0,C 180,E1 -2954.644,E2 -2954.644} C_VEL
LIN {X 0,Y 560.474,Z 446.721,A -85,B 0,C 180,E1 -2954.961,E2 -2954.961} C_VEL
LIN {X 0,Y 560.311,Z 460.499,A -85,B 0,C 180,E1 -2955.422,E2 -2955.422} C_VEL
LIN {X 0,Y 560.105,Z 473.881,A -85,B 0,C 180,E1 -2956.023,E2 -2956.023} C_VEL
LIN {X 0,Y 559.81,Z 486.68,A -85,B 0,C 180,E1 -2956.755,E2 -2956.755} C_VEL
LIN {X 0,Y 559.636,Z 498.314,A -85,B 0,C 180,E1 -2957.581,E2 -2957.581} C_VEL
LIN {X 0,Y 559.437,Z 508.887,A -85,B 0,C 180,E1 -2958.489,E2 -2958.489} C_VEL
LIN {X 0,Y 559.272,Z 518.709,A -85,B 0,C 180,E1 -2959.502,E2 -2959.502} C_VEL
LIN {X 0,Y 559.121,Z 527.559,A -85,B 0,C 180,E1 -2960.596,E2 -2960.596} C_VEL
LIN {X 0,Y 558.986,Z 536.036,A -85,B 0,C 180,E1 -2961.869,E2 -2961.869} C_VEL
LIN {X 0,Y 558.901,Z 542.866,A -85,B 0,C 180,E1 -2963.14,E2 -2963.14} C_VEL
LIN {X 0,Y 558.913,Z 547.57,A -85,B 0,C 180,E1 -2964.227,E2 -2964.227} C_VEL
LIN {X 0,Y 558.865,Z 552.444,A -85,B 0,C 180,E1 -2965.673,E2 -2965.673} C_VEL
LIN {X 0,Y 558.796,Z 555.832,A -85,B 0,C 180,E1 -2967.116,E2 -2967.116} C_VEL
LIN {X 0,Y 558.74,Z 557.834,A -85,B 0,C 180,E1 -2968.559,E2 -2968.559} C_VEL
LIN {X 0,Y 558.738,Z 558.5,A -85,B 0,C 180,E1 -2970,E2 -2970} C_VEL
LIN {X 0,Y 558.74,Z 557.835,A -85,B 0,C 180,E1 -2971.442,E2 -2971.442} C_VEL
LIN {X 0,Y 558.796,Z 555.835,A -85,B 0,C 180,E1 -2972.884,E2 -2972.884} C_VEL
LIN {X 0,Y 558.865,Z 552.446,A -85,B 0,C 180,E1 -2974.327,E2 -2974.327} C_VEL
LIN {X 0,Y 558.914,Z 547.568,A -85,B 0,C 180,E1 -2975.773,E2 -2975.773} C_VEL
LIN {X 0,Y 558.906,Z 541.055,A -85,B 0,C 180,E1 -2977.224,E2 -2977.224} C_VEL
LIN {X 0,Y 559.028,Z 533.803,A -85,B 0,C 180,E1 -2978.495,E2 -2978.495} C_VEL
LIN {X 0,Y 559.146,Z 524.823,A -85,B 0,C 180,E1 -2979.769,E2 -2979.769} C_VEL
LIN {X 0,Y 559.35,Z 515.394,A -85,B 0,C 180,E1 -2980.863,E2 -2980.863} C_VEL
LIN {X 0,Y 559.518,Z 504.956,A -85,B 0,C 180,E1 -2981.869,E2 -2981.869} C_VEL
LIN {X 0,Y 559.708,Z 493.434,A -85,B 0,C 180,E1 -2982.786,E2 -2982.786} C_VEL
LIN {X 0,Y 559.923,Z 480.644,A -85,B 0,C 180,E1 -2983.612,E2 -2983.612} C_VEL
LIN {X 0,Y 560.166,Z 468.153,A -85,B 0,C 180,E1 -2984.254,E2 -2984.254} C_VEL
LIN {X 0,Y 560.405,Z 454.992,A -85,B 0,C 180,E1 -2984.778,E2 -2984.778} C_VEL
LIN {X 0,Y 560.545,Z 441.494,A -85,B 0,C 180,E1 -2985.171,E2 -2985.171} C_VEL
LIN {X 0,Y 560.612,Z 426.622,A -85,B 0,C 180,E1 -2985.45,E2 -2985.45} C_VEL
LIN {X 0,Y 560.886,Z 302.57,A -85,B 0,C 180,E1 -2987.063,E2 -2987.063} C_VEL
LIN {X 0,Y 559.696,Z 296.21,A -85,B 0,C 180,E1 -2987.2,E2 -2987.2} C_VEL
LIN {X 0,Y 559.695,Z 292.128,A -85,B 0,C 180,E1 -2987.728,E2 -2987.728} C_VEL
LIN {X 0,Y 560.09,Z 270.572,A -85,B 0,C 180,E1 -2990.761,E2 -2990.761} C_VEL
LIN {X 0,Y 560.329,Z 254.546,A -85,B 0,C 180,E1 -2993.054,E2 -2993.054} C_VEL
LIN {X 0,Y 559.216,Z 248.59,A -85,B 0,C 180,E1 -2994.008,E2 -2994.008} C_VEL
LIN {X 0,Y 559.169,Z 248.458,A -85,B 0,C 180,E1 -2996.902,E2 -2996.902} C_VEL
LIN {X 0,Y 559.148,Z 248.449,A -85,B 0,C 180,E1 -2999.857,E2 -2999.857} C_VEL
LIN {X 0,Y 559.174,Z 248.457,A -85,B 0,C 180,E1 -3002.713,E2 -3002.713} C_VEL
LIN {X 0,Y 559.126,Z 248.459,A -85,B 0,C 180,E1 -3005.323,E2 -3005.323} C_VEL
LIN {X 0,Y 559.13,Z 248.458,A -85,B 0,C 180,E1 -3008.017,E2 -3008.017} C_VEL
LIN {X 0,Y 559.155,Z 248.454,A -85,B 0,C 180,E1 -3010.811,E2 -3010.811} C_VEL
LIN {X 0,Y 559.159,Z 248.455,A -85,B 0,C 180,E1 -3013.731,E2 -3013.731} C_VEL
LIN {X 0,Y 559.141,Z 248.458,A -85,B 0,C 180,E1 -3016.803,E2 -3016.803} C_VEL
LIN {X 0,Y 559.17,Z 248.451,A -85,B 0,C 180,E1 -3019.189,E2 -3019.189} C_VEL
LIN {X 0,Y 559.13,Z 248.463,A -85,B 0,C 180,E1 -3021.982,E2 -3021.982} C_VEL
LIN {X 0,Y 559.154,Z 248.448,A -85,B 0,C 180,E1 -3024.782,E2 -3024.782} C_VEL
LIN {X 0,Y 559.167,Z 248.449,A -85,B 0,C 180,E1 -3027.361,E2 -3027.361} C_VEL
LIN {X 0,Y 559.182,Z 248.459,A -85,B 0,C 180,E1 -3030.135,E2 -3030.135} C_VEL
LIN {X 0,Y 559.176,Z 248.45,A -85,B 0,C 180,E1 -3033.169,E2 -3033.169} C_VEL
LIN {X 0,Y 559.15,Z 248.458,A -85,B 0,C 180,E1 -3035.495,E2 -3035.495} C_VEL
LIN {X 0,Y 559.163,Z 248.453,A -85,B 0,C 180,E1 -3038.624,E2 -3038.624} C_VEL
LIN {X 0,Y 559.163,Z 248.453,A -85,B 0,C 180,E1 -3040.926,E2 -3040.926} C_VEL
LIN {X 0,Y 559.164,Z 248.459,A -85,B 0,C 180,E1 -3043.948,E2 -3043.948} C_VEL
LIN {X 0,Y 559.167,Z 248.456,A -85,B 0,C 180,E1 -3046.184,E2 -3046.184} C_VEL
LIN {X 0,Y 559.186,Z 248.45,A -85,B 0,C 180,E1 -3049.133,E2 -3049.133} C_VEL
LIN {X 0,Y 559.199,Z 248.452,A -85,B 0,C 180,E1 -3052.054,E2 -3052.054} C_VEL
LIN {X 0,Y 559.249,Z 248.442,A -85,B 0,C 180,E1 -3054.953,E2 -3054.953} C_VEL
LIN {X 0,Y 559.244,Z 248.448,A -85,B 0,C 180,E1 -3057.839,E2 -3057.839} C_VEL
LIN {X 0,Y 559.267,Z 248.44,A -85,B 0,C 180,E1 -3060.72,E2 -3060.72} C_VEL
LIN {X 0,Y 559.236,Z 248.442,A -85,B 0,C 180,E1 -3062.881,E2 -3062.881} C_VEL
LIN {X 0,Y 559.223,Z 248.449,A -85,B 0,C 180,E1 -3065.77,E2 -3065.77} C_VEL
LIN {X 0,Y 559.185,Z 248.449,A -85,B 0,C 180,E1 -3068.674,E2 -3068.674} C_VEL
LIN {X 0,Y 559.196,Z 248.454,A -85,B 0,C 180,E1 -3071.601,E2 -3071.601} C_VEL
LIN {X 0,Y 559.191,Z 248.449,A -85,B 0,C 180,E1 -3074.596,E2 -3074.596} C_VEL
LIN {X 0,Y 559.156,Z 248.458,A -85,B 0,C 180,E1 -3077.557,E2 -3077.557} C_VEL
LIN {X 0,Y 559.165,Z 248.452,A -85,B 0,C 180,E1 -3079.838,E2 -3079.838} C_VEL
LIN {X 0,Y 559.134,Z 248.456,A -85,B 0,C 180,E1 -3082.153,E2 -3082.153} C_VEL
LIN {X 0,Y 559.172,Z 248.457,A -85,B 0,C 180,E1 -3085.188,E2 -3085.188} C_VEL
LIN {X 0,Y 559.186,Z 248.451,A -85,B 0,C 180,E1 -3087.712,E2 -3087.712} C_VEL
LIN {X 0,Y 559.147,Z 248.456,A -85,B 0,C 180,E1 -3090.626,E2 -3090.626} C_VEL
LIN {X 0,Y 558.483,Z 248.541,A -85,B 0,C 180,E1 -3091.227,E2 -3091.227} C_VEL
LIN {X 0,Y 555.618,Z 248.894,A -85,B 0,C 180,E1 -3092.203,E2 -3092.203} C_VEL
LIN {X 0,Y 553.205,Z 249.193,A -85,B 0,C 180,E1 -3092.989,E2 -3092.989} C_VEL
LIN {X 0,Y 552.184,Z 249.315,A -85,B 0,C 180,E1 -3093.596,E2 -3093.596} C_VEL
LIN {X 0,Y 552.11,Z 249.323,A -85,B 0,C 180,E1 -3093.801,E2 -3093.801} C_VEL
LIN {X 0,Y 552.107,Z 249.338,A -85,B 0,C 180,E1 -3096.747,E2 -3096.747} C_VEL
LIN {X 0,Y 552.13,Z 249.328,A -85,B 0,C 180,E1 -3099.527,E2 -3099.527} C_VEL
LIN {X 0,Y 552.126,Z 249.328,A -85,B 0,C 180,E1 -3102.426,E2 -3102.426} C_VEL
LIN {X 0,Y 552.096,Z 249.333,A -85,B 0,C 180,E1 -3105.564,E2 -3105.564} C_VEL
LIN {X 0,Y 552.138,Z 249.334,A -85,B 0,C 180,E1 -3108.677,E2 -3108.677} C_VEL
LIN {X 0,Y 552.116,Z 249.33,A -85,B 0,C 180,E1 -3111.412,E2 -3111.412} C_VEL
LIN {X 0,Y 552.101,Z 249.337,A -85,B 0,C 180,E1 -3114.158,E2 -3114.158} C_VEL
LIN {X 0,Y 552.122,Z 249.335,A -85,B 0,C 180,E1 -3116.815,E2 -3116.815} C_VEL
LIN {X 0,Y 552.102,Z 249.334,A -85,B 0,C 180,E1 -3119.391,E2 -3119.391} C_VEL
LIN {X 0,Y 552.12,Z 249.33,A -85,B 0,C 180,E1 -3121.903,E2 -3121.903} C_VEL
LIN {X 0,Y 552.157,Z 249.326,A -85,B 0,C 180,E1 -3124.65,E2 -3124.65} C_VEL
LIN {X 0,Y 552.151,Z 249.468,A -85,B 0,C 180,E1 -3126.934,E2 -3126.934} C_VEL
LIN {X 0,Y 553.216,Z 255.068,A -85,B 0,C 180,E1 -3127.874,E2 -3127.874} C_VEL
LIN {X 0,Y 552.889,Z 273.563,A -85,B 0,C 180,E1 -3130.701,E2 -3130.701} C_VEL
LIN {X 0,Y 552.695,Z 286.409,A -85,B 0,C 180,E1 -3132.609,E2 -3132.609} C_VEL
LIN {X 0,Y 553.586,Z 291.301,A -85,B 0,C 180,E1 -3132.733,E2 -3132.733} C_VEL
LIN {X 0,Y 554.215,Z 296.045,A -85,B 0,C 180,E1 -3132.816,E2 -3132.816} C_VEL
LIN {X 0,Y 553.784,Z 422.78,A -85,B 0,C 180,E1 -3134.497,E2 -3134.497} C_VEL
LIN {X 0,Y 553.556,Z 437.518,A -85,B 0,C 180,E1 -3134.838,E2 -3134.838} C_VEL
LIN {X 0,Y 553.358,Z 451.748,A -85,B 0,C 180,E1 -3135.332,E2 -3135.332} C_VEL
LIN {X 0,Y 553.168,Z 464.795,A -85,B 0,C 180,E1 -3135.938,E2 -3135.938} C_VEL
LIN {X 0,Y 552.912,Z 477.419,A -85,B 0,C 180,E1 -3136.681,E2 -3136.681} C_VEL
LIN {X 0,Y 552.641,Z 488.917,A -85,B 0,C 180,E1 -3137.515,E2 -3137.515} C_VEL
LIN {X 0,Y 552.45,Z 498.981,A -85,B 0,C 180,E1 -3138.396,E2 -3138.396} C_VEL
LIN {X 0,Y 552.286,Z 508.313,A -85,B 0,C 180,E1 -3139.367,E2 -3139.367} C_VEL
LIN {X 0,Y 552.074,Z 517.228,A -85,B 0,C 180,E1 -3140.474,E2 -3140.474} C_VEL
LIN {X 0,Y 551.928,Z 525.764,A -85,B 0,C 180,E1 -3141.764,E2 -3141.764} C_VEL
LIN {X 0,Y 551.824,Z 532.641,A -85,B 0,C 180,E1 -3143.051,E2 -3143.051} C_VEL
LIN {X 0,Y 551.792,Z 538.804,A -85,B 0,C 180,E1 -3144.519,E2 -3144.519} C_VEL
LIN {X 0,Y 551.76,Z 542.316,A -85,B 0,C 180,E1 -3145.617,E2 -3145.617} C_VEL
LIN {X 0,Y 551.72,Z 545.747,A -85,B 0,C 180,E1 -3147.079,E2 -3147.079} C_VEL
LIN {X 0,Y 551.643,Z 547.787,A -85,B 0,C 180,E1 -3148.54,E2 -3148.54} C_VEL
LIN {X 0,Y 551.64,Z 548.496,A -85,B 0,C 180,E1 -3150,E2 -3150} C_VEL
LIN {X 0,Y 551.641,Z 547.879,A -85,B 0,C 180,E1 -3151.46,E2 -3151.46} C_VEL
LIN {X 0,Y 551.719,Z 545.921,A -85,B 0,C 180,E1 -3152.921,E2 -3152.921} C_VEL
LIN {X 0,Y 551.76,Z 542.575,A -85,B 0,C 180,E1 -3154.383,E2 -3154.383} C_VEL
LIN {X 0,Y 551.819,Z 537.744,A -85,B 0,C 180,E1 -3155.848,E2 -3155.848} C_VEL
LIN {X 0,Y 551.833,Z 531.277,A -85,B 0,C 180,E1 -3157.317,E2 -3157.317} C_VEL
LIN {X 0,Y 551.962,Z 524.077,A -85,B 0,C 180,E1 -3158.604,E2 -3158.604} C_VEL
LIN {X 0,Y 552.067,Z 516.534,A -85,B 0,C 180,E1 -3159.711,E2 -3159.711} C_VEL
LIN {X 0,Y 552.282,Z 507.476,A -85,B 0,C 180,E1 -3160.818,E2 -3160.818} C_VEL
LIN {X 0,Y 552.481,Z 496.51,A -85,B 0,C 180,E1 -3161.929,E2 -3161.929} C_VEL
LIN {X 0,Y 552.719,Z 485.336,A -85,B 0,C 180,E1 -3162.857,E2 -3162.857} C_VEL
LIN {X 0,Y 553,Z 472.982,A -85,B 0,C 180,E1 -3163.692,E2 -3163.692} C_VEL
LIN {X 0,Y 553.238,Z 461.096,A -85,B 0,C 180,E1 -3164.342,E2 -3164.342} C_VEL
LIN {X 0,Y 553.486,Z 448.242,A -85,B 0,C 180,E1 -3164.894,E2 -3164.894} C_VEL
LIN {X 0,Y 553.629,Z 434.191,A -85,B 0,C 180,E1 -3165.341,E2 -3165.341} C_VEL
LIN {X 0,Y 553.772,Z 419.512,A -85,B 0,C 180,E1 -3165.645,E2 -3165.645} C_VEL
LIN {X 0,Y 554.16,Z 294.286,A -85,B 0,C 180,E1 -3167.299,E2 -3167.299} C_VEL
LIN {X 0,Y 552.721,Z 286.614,A -85,B 0,C 180,E1 -3167.466,E2 -3167.466} C_VEL
LIN {X 0,Y 552.841,Z 275.435,A -85,B 0,C 180,E1 -3169.107,E2 -3169.107} C_VEL
LIN {X 0,Y 553.249,Z 255.804,A -85,B 0,C 180,E1 -3172.1,E2 -3172.1} C_VEL
LIN {X 0,Y 552.114,Z 249.392,A -85,B 0,C 180,E1 -3173.191,E2 -3173.191} C_VEL
LIN {X 0,Y 552.131,Z 249.332,A -85,B 0,C 180,E1 -3175.644,E2 -3175.644} C_VEL
LIN {X 0,Y 552.124,Z 249.327,A -85,B 0,C 180,E1 -3178.561,E2 -3178.561} C_VEL
LIN {X 0,Y 552.11,Z 249.338,A -85,B 0,C 180,E1 -3181.475,E2 -3181.475} C_VEL
LIN {X 0,Y 552.133,Z 249.33,A -85,B 0,C 180,E1 -3184.17,E2 -3184.17} C_VEL
LIN {X 0,Y 552.107,Z 249.333,A -85,B 0,C 180,E1 -3186.746,E2 -3186.746} C_VEL
LIN {X 0,Y 552.128,Z 249.339,A -85,B 0,C 180,E1 -3189.526,E2 -3189.526} C_VEL
LIN {X 0,Y 552.127,Z 249.325,A -85,B 0,C 180,E1 -3192.425,E2 -3192.425} C_VEL
LIN {X 0,Y 552.093,Z 249.34,A -85,B 0,C 180,E1 -3195.562,E2 -3195.562} C_VEL
LIN {X 0,Y 552.133,Z 249.324,A -85,B 0,C 180,E1 -3198.676,E2 -3198.676} C_VEL
LIN {X 0,Y 552.115,Z 249.339,A -85,B 0,C 180,E1 -3201.411,E2 -3201.411} C_VEL
LIN {X 0,Y 552.108,Z 249.331,A -85,B 0,C 180,E1 -3204.158,E2 -3204.158} C_VEL
LIN {X 0,Y 552.116,Z 249.327,A -85,B 0,C 180,E1 -3206.814,E2 -3206.814} C_VEL
LIN {X 0,Y 552.107,Z 249.337,A -85,B 0,C 180,E1 -3209.391,E2 -3209.391} C_VEL
LIN {X 0,Y 552.118,Z 249.331,A -85,B 0,C 180,E1 -3211.902,E2 -3211.902} C_VEL
LIN {X 0,Y 552.147,Z 249.328,A -85,B 0,C 180,E1 -3214.649,E2 -3214.649} C_VEL
LIN {X 0,Y 552.088,Z 249.335,A -85,B 0,C 180,E1 -3217.549,E2 -3217.549} C_VEL
LIN {X 0,Y 552.14,Z 249.328,A -85,B 0,C 180,E1 -3220.373,E2 -3220.373} C_VEL
LIN {X 0,Y 552.149,Z 249.333,A -85,B 0,C 180,E1 -3222.977,E2 -3222.977} C_VEL
LIN {X 0,Y 552.129,Z 249.327,A -85,B 0,C 180,E1 -3226.004,E2 -3226.004} C_VEL
LIN {X 0,Y 552.169,Z 249.329,A -85,B 0,C 180,E1 -3228.993,E2 -3228.993} C_VEL
LIN {X 0,Y 552.152,Z 249.324,A -85,B 0,C 180,E1 -3231.951,E2 -3231.951} C_VEL
LIN {X 0,Y 552.224,Z 249.322,A -85,B 0,C 180,E1 -3234.889,E2 -3234.889} C_VEL
LIN {X 0,Y 552.214,Z 249.315,A -85,B 0,C 180,E1 -3237.812,E2 -3237.812} C_VEL
LIN {X 0,Y 552.238,Z 249.322,A -85,B 0,C 180,E1 -3240.729,E2 -3240.729} C_VEL
LIN {X 0,Y 552.202,Z 249.32,A -85,B 0,C 180,E1 -3242.918,E2 -3242.918} C_VEL
LIN {X 0,Y 552.192,Z 249.322,A -85,B 0,C 180,E1 -3245.844,E2 -3245.844} C_VEL
LIN {X 0,Y 552.162,Z 249.326,A -85,B 0,C 180,E1 -3248.786,E2 -3248.786} C_VEL
LIN {X 0,Y 552.153,Z 249.326,A -85,B 0,C 180,E1 -3251.751,E2 -3251.751} C_VEL
LIN {X 0,Y 552.127,Z 249.331,A -85,B 0,C 180,E1 -3254.749,E2 -3254.749} C_VEL
LIN {X 0,Y 552.106,Z 249.333,A -85,B 0,C 180,E1 -3257.789,E2 -3257.789} C_VEL
LIN {X 0,Y 552.123,Z 249.339,A -85,B 0,C 180,E1 -3260.101,E2 -3260.101} C_VEL
LIN {X 0,Y 552.088,Z 249.337,A -85,B 0,C 180,E1 -3262.451,E2 -3262.451} C_VEL
LIN {X 0,Y 552.147,Z 249.328,A -85,B 0,C 180,E1 -3265.351,E2 -3265.351} C_VEL
LIN {X 0,Y 552.118,Z 249.338,A -85,B 0,C 180,E1 -3268.098,E2 -3268.098} C_VEL
LIN {X 0,Y 552.107,Z 249.333,A -85,B 0,C 180,E1 -3270.609,E2 -3270.609} C_VEL
LIN {X 0,Y 552.116,Z 249.327,A -85,B 0,C 180,E1 -3273.186,E2 -3273.186} C_VEL
LIN {X 0,Y 552.107,Z 249.334,A -85,B 0,C 180,E1 -3275.842,E2 -3275.842} C_VEL
LIN {X 0,Y 552.12,Z 249.331,A -85,B 0,C 180,E1 -3279.063,E2 -3279.063} C_VEL
LIN {X 0,Y 552.134,Z 249.332,A -85,B 0,C 180,E1 -3281.445,E2 -3281.445} C_VEL
LIN {X 0,Y 552.09,Z 249.334,A -85,B 0,C 180,E1 -3284.533,E2 -3284.533} C_VEL
LIN {X 0,Y 552.127,Z 249.335,A -85,B 0,C 180,E1 -3287.585,E2 -3287.585} C_VEL
LIN {X 0,Y 552.13,Z 249.33,A -85,B 0,C 180,E1 -3290.474,E2 -3290.474} C_VEL
LIN {X 0,Y 552.103,Z 249.336,A -85,B 0,C 180,E1 -3293.318,E2 -3293.318} C_VEL
LIN {X 0,Y 552.126,Z 249.331,A -85,B 0,C 180,E1 -3295.94,E2 -3295.94} C_VEL
LIN {X 0,Y 552.117,Z 249.331,A -85,B 0,C 180,E1 -3298.541,E2 -3298.541} C_VEL
LIN {X 0,Y 552.123,Z 249.334,A -85,B 0,C 180,E1 -3301.439,E2 -3301.439} C_VEL
LIN {X 0,Y 552.13,Z 249.328,A -85,B 0,C 180,E1 -3304.356,E2 -3304.356} C_VEL
LIN {X 0,Y 552.156,Z 249.492,A -85,B 0,C 180,E1 -3305.815,E2 -3305.815} C_VEL
LIN {X 0,Y 553.373,Z 255.686,A -85,B 0,C 180,E1 -3306.815,E2 -3306.815} C_VEL
LIN {X 0,Y 553.107,Z 270.51,A -85,B 0,C 180,E1 -3308.964,E2 -3308.964} C_VEL
LIN {X 0,Y 552.789,Z 290.725,A -85,B 0,C 180,E1 -3311.852,E2 -3311.852} C_VEL
LIN {X 0,Y 552.698,Z 295.934,A -85,B 0,C 180,E1 -3312.562,E2 -3312.562} C_VEL
LIN {X 0,Y 553.697,Z 301.529,A -85,B 0,C 180,E1 -3312.695,E2 -3312.695} C_VEL
LIN {X 0,Y 554.244,Z 306.167,A -85,B 0,C 180,E1 -3312.775,E2 -3312.775} C_VEL
LIN {X 0,Y 553.778,Z 432.657,A -85,B 0,C 180,E1 -3314.449,E2 -3314.449} C_VEL
LIN {X 0,Y 553.605,Z 447.274,A -85,B 0,C 180,E1 -3314.787,E2 -3314.787} C_VEL
LIN {X 0,Y 553.37,Z 461.713,A -85,B 0,C 180,E1 -3315.286,E2 -3315.286} C_VEL
LIN {X 0,Y 553.166,Z 475.644,A -85,B 0,C 180,E1 -3315.938,E2 -3315.938} C_VEL
LIN {X 0,Y 552.863,Z 488.103,A -85,B 0,C 180,E1 -3316.679,E2 -3316.679} C_VEL
LIN {X 0,Y 552.617,Z 500.652,A -85,B 0,C 180,E1 -3317.608,E2 -3317.608} C_VEL
LIN {X 0,Y 552.45,Z 511.277,A -85,B 0,C 180,E1 -3318.571,E2 -3318.571} C_VEL
LIN {X 0,Y 552.179,Z 521.854,A -85,B 0,C 180,E1 -3319.736,E2 -3319.736} C_VEL
LIN {X 0,Y 552.032,Z 530.176,A -85,B 0,C 180,E1 -3320.843,E2 -3320.843} C_VEL
LIN {X 0,Y 551.913,Z 538.128,A -85,B 0,C 180,E1 -3322.132,E2 -3322.132} C_VEL
LIN {X 0,Y 551.821,Z 544.529,A -85,B 0,C 180,E1 -3323.418,E2 -3323.418} C_VEL
LIN {X 0,Y 551.792,Z 548.961,A -85,B 0,C 180,E1 -3324.519,E2 -3324.519} C_VEL
LIN {X 0,Y 551.759,Z 552.444,A -85,B 0,C 180,E1 -3325.617,E2 -3325.617} C_VEL
LIN {X 0,Y 551.72,Z 555.832,A -85,B 0,C 180,E1 -3327.079,E2 -3327.079} C_VEL
LIN {X 0,Y 551.64,Z 557.834,A -85,B 0,C 180,E1 -3328.54,E2 -3328.54} C_VEL
LIN {X 0,Y 551.639,Z 558.5,A -85,B 0,C 180,E1 -3330,E2 -3330} C_VEL
LIN {X 0,Y 551.64,Z 557.835,A -85,B 0,C 180,E1 -3331.46,E2 -3331.46} C_VEL
LIN {X 0,Y 551.72,Z 555.835,A -85,B 0,C 180,E1 -3332.921,E2 -3332.921} C_VEL
LIN {X 0,Y 551.759,Z 552.447,A -85,B 0,C 180,E1 -3334.383,E2 -3334.383} C_VEL
LIN {X 0,Y 551.823,Z 547.568,A -85,B 0,C 180,E1 -3335.848,E2 -3335.848} C_VEL
LIN {X 0,Y 551.832,Z 541.055,A -85,B 0,C 180,E1 -3337.317,E2 -3337.317} C_VEL
LIN {X 0,Y 551.962,Z 533.804,A -85,B 0,C 180,E1 -3338.604,E2 -3338.604} C_VEL
LIN {X 0,Y 552.116,Z 524.823,A -85,B 0,C 180,E1 -3339.895,E2 -3339.895} C_VEL
LIN {X 0,Y 552.346,Z 515.394,A -85,B 0,C 180,E1 -3341.003,E2 -3341.003} C_VEL
LIN {X 0,Y 552.539,Z 504.955,A -85,B 0,C 180,E1 -3342.021,E2 -3342.021} C_VEL
LIN {X 0,Y 552.76,Z 493.431,A -85,B 0,C 180,E1 -3342.949,E2 -3342.949} C_VEL
LIN {X 0,Y 553.012,Z 480.642,A -85,B 0,C 180,E1 -3343.785,E2 -3343.785} C_VEL
LIN {X 0,Y 553.283,Z 468.15,A -85,B 0,C 180,E1 -3344.435,E2 -3344.435} C_VEL
LIN {X 0,Y 553.506,Z 454.858,A -85,B 0,C 180,E1 -3344.971,E2 -3344.971} C_VEL
LIN {X 0,Y 553.7,Z 440.862,A -85,B 0,C 180,E1 -3345.38,E2 -3345.38} C_VEL
LIN {X 0,Y 553.78,Z 426.622,A -85,B 0,C 180,E1 -3345.645,E2 -3345.645} C_VEL
LIN {X 0,Y 554.143,Z 303.659,A -85,B 0,C 180,E1 -3347.262,E2 -3347.262} C_VEL
LIN {X 0,Y 552.727,Z 296.202,A -85,B 0,C 180,E1 -3347.421,E2 -3347.421} C_VEL
LIN {X 0,Y 552.741,Z 292.072,A -85,B 0,C 180,E1 -3347.959,E2 -3347.959} C_VEL
LIN {X 0,Y 553.151,Z 271.861,A -85,B 0,C 180,E1 -3350.839,E2 -3350.839} C_VEL
LIN {X 0,Y 553.371,Z 255.686,A -85,B 0,C 180,E1 -3353.185,E2 -3353.185} C_VEL
LIN {X 0,Y 552.157,Z 249.499,A -85,B 0,C 180,E1 -3354.185,E2 -3354.185} C_VEL
LIN {X 0,Y 552.139,Z 249.335,A -85,B 0,C 180,E1 -3357,E2 -3357} C_VEL
LIN {X 0,Y 552.116,Z 249.325,A -85,B 0,C 180,E1 -3360.05,E2 -3360.05} C_VEL
LIN {X 0,Y 552.127,Z 249.333,A -85,B 0,C 180,E1 -3362.848,E2 -3362.848} C_VEL
LIN {X 0,Y 552.075,Z 249.337,A -85,B 0,C 180,E1 -3365.439,E2 -3365.439} C_VEL
LIN {X 0,Y 552.093,Z 249.333,A -85,B 0,C 180,E1 -3367.885,E2 -3367.885} C_VEL
LIN {X 0,Y 552.107,Z 249.336,A -85,B 0,C 180,E1 -3370.48,E2 -3370.48} C_VEL
LIN {X 0,Y 552.111,Z 249.331,A -85,B 0,C 180,E1 -3373.484,E2 -3373.484} C_VEL
LIN {X 0,Y 552.102,Z 249.338,A -85,B 0,C 180,E1 -3376.576,E2 -3376.576} C_VEL
LIN {X 0,Y 552.116,Z 249.33,A -85,B 0,C 180,E1 -3379.519,E2 -3379.519} C_VEL
LIN {X 0,Y 552.089,Z 249.34,A -85,B 0,C 180,E1 -3382.336,E2 -3382.336} C_VEL
LIN {X 0,Y 552.123,Z 249.321,A -85,B 0,C 180,E1 -3385.054,E2 -3385.054} C_VEL
LIN {X 0,Y 552.121,Z 249.329,A -85,B 0,C 180,E1 -3387.682,E2 -3387.682} C_VEL
LIN {X 0,Y 552.138,Z 249.334,A -85,B 0,C 180,E1 -3390.237,E2 -3390.237} C_VEL
LIN {X 0,Y 552.141,Z 249.326,A -85,B 0,C 180,E1 -3392.997,E2 -3392.997} C_VEL
LIN {X 0,Y 552.106,Z 249.333,A -85,B 0,C 180,E1 -3395.161,E2 -3395.161} C_VEL
LIN {X 0,Y 552.088,Z 249.337,A -85,B 0,C 180,E1 -3397.549,E2 -3397.549} C_VEL
LIN {X 0,Y 552.149,Z 249.327,A -85,B 0,C 180,E1 -3400.674,E2 -3400.674} C_VEL
LIN {X 0,Y 552.113,Z 249.337,A -85,B 0,C 180,E1 -3403.737,E2 -3403.737} C_VEL
LIN {X 0,Y 552.129,Z 249.335,A -85,B 0,C 180,E1 -3406.004,E2 -3406.004} C_VEL
LIN {X 0,Y 552.154,Z 249.325,A -85,B 0,C 180,E1 -3408.993,E2 -3408.993} C_VEL
LIN {X 0,Y 552.152,Z 249.331,A -85,B 0,C 180,E1 -3411.951,E2 -3411.951} C_VEL
LIN {X 0,Y 552.223,Z 249.317,A -85,B 0,C 180,E1 -3414.889,E2 -3414.889} C_VEL
LIN {X 0,Y 552.215,Z 249.324,A -85,B 0,C 180,E1 -3417.812,E2 -3417.812} C_VEL
LIN {X 0,Y 552.237,Z 249.316,A -85,B 0,C 180,E1 -3420.729,E2 -3420.729} C_VEL
LIN {X 0,Y 552.202,Z 249.318,A -85,B 0,C 180,E1 -3422.918,E2 -3422.918} C_VEL
LIN {X 0,Y 552.193,Z 249.324,A -85,B 0,C 180,E1 -3425.844,E2 -3425.844} C_VEL
LIN {X 0,Y 552.156,Z 249.325,A -85,B 0,C 180,E1 -3428.786,E2 -3428.786} C_VEL
LIN {X 0,Y 552.154,Z 249.329,A -85,B 0,C 180,E1 -3431.751,E2 -3431.751} C_VEL
LIN {X 0,Y 552.128,Z 249.33,A -85,B 0,C 180,E1 -3434.749,E2 -3434.749} C_VEL
LIN {X 0,Y 552.107,Z 249.334,A -85,B 0,C 180,E1 -3437.789,E2 -3437.789} C_VEL
LIN {X 0,Y 552.123,Z 249.328,A -85,B 0,C 180,E1 -3440.102,E2 -3440.102} C_VEL
LIN {X 0,Y 552.088,Z 249.334,A -85,B 0,C 180,E1 -3442.451,E2 -3442.451} C_VEL
LIN {X 0,Y 552.148,Z 249.329,A -85,B 0,C 180,E1 -3445.351,E2 -3445.351} C_VEL
LIN {X 0,Y 552.119,Z 249.33,A -85,B 0,C 180,E1 -3448.098,E2 -3448.098} C_VEL
LIN {X 0,Y 552.107,Z 249.336,A -85,B 0,C 180,E1 -3450.621,E2 -3450.621} C_VEL
LIN {X 0,Y 552.117,Z 249.327,A -85,B 0,C 180,E1 -3453.186,E2 -3453.186} C_VEL
LIN {X 0,Y 552.11,Z 249.323,A -85,B 0,C 180,E1 -3453.801,E2 -3453.801} C_VEL
LIN {X 0,Y 551.475,Z 249.405,A -85,B 0,C 180,E1 -3454.41,E2 -3454.41} C_VEL
LIN {X 0,Y 548.653,Z 249.768,A -85,B 0,C 180,E1 -3455.398,E2 -3455.398} C_VEL
LIN {X 0,Y 546.231,Z 250.076,A -85,B 0,C 180,E1 -3456.193,E2 -3456.193} C_VEL
LIN {X 0,Y 545.162,Z 250.207,A -85,B 0,C 180,E1 -3456.807,E2 -3456.807} C_VEL
LIN {X 0,Y 545.06,Z 250.217,A -85,B 0,C 180,E1 -3457.015,E2 -3457.015} C_VEL
LIN {X 0,Y 545.07,Z 250.208,A -85,B 0,C 180,E1 -3460.142,E2 -3460.142} C_VEL
LIN {X 0,Y 545.074,Z 250.211,A -85,B 0,C 180,E1 -3463.107,E2 -3463.107} C_VEL
LIN {X 0,Y 545.062,Z 250.213,A -85,B 0,C 180,E1 -3466.225,E2 -3466.225} C_VEL
LIN {X 0,Y 545.095,Z 250.211,A -85,B 0,C 180,E1 -3468.888,E2 -3468.888} C_VEL
LIN {X 0,Y 545.05,Z 250.21,A -85,B 0,C 180,E1 -3471.763,E2 -3471.763} C_VEL
LIN {X 0,Y 545.052,Z 250.219,A -85,B 0,C 180,E1 -3474.534,E2 -3474.534} C_VEL
LIN {X 0,Y 545.081,Z 250.209,A -85,B 0,C 180,E1 -3477.213,E2 -3477.213} C_VEL
LIN {X 0,Y 545.063,Z 250.212,A -85,B 0,C 180,E1 -3479.811,E2 -3479.811} C_VEL
LIN {X 0,Y 545.089,Z 250.207,A -85,B 0,C 180,E1 -3482.345,E2 -3482.345} C_VEL
LIN {X 0,Y 545.118,Z 250.201,A -85,B 0,C 180,E1 -3484.821,E2 -3484.821} C_VEL
LIN {X 0,Y 545.123,Z 250.434,A -85,B 0,C 180,E1 -3486.77,E2 -3486.77} C_VEL
LIN {X 0,Y 546.32,Z 256.875,A -85,B 0,C 180,E1 -3487.855,E2 -3487.855} C_VEL
LIN {X 0,Y 545.937,Z 274.892,A -85,B 0,C 180,E1 -3490.641,E2 -3490.641} C_VEL
LIN {X 0,Y 545.73,Z 286.482,A -85,B 0,C 180,E1 -3492.381,E2 -3492.381} C_VEL
LIN {X 0,Y 546.605,Z 291.039,A -85,B 0,C 180,E1 -3492.5,E2 -3492.5} C_VEL
LIN {X 0,Y 547.456,Z 297.071,A -85,B 0,C 180,E1 -3492.609,E2 -3492.609} C_VEL
LIN {X 0,Y 546.957,Z 422.881,A -85,B 0,C 180,E1 -3494.298,E2 -3494.298} C_VEL
LIN {X 0,Y 546.718,Z 437.599,A -85,B 0,C 180,E1 -3494.644,E2 -3494.644} C_VEL
LIN {X 0,Y 546.492,Z 451.814,A -85,B 0,C 180,E1 -3495.144,E2 -3495.144} C_VEL
LIN {X 0,Y 546.271,Z 464.845,A -85,B 0,C 180,E1 -3495.756,E2 -3495.756} C_VEL
LIN {X 0,Y 545.963,Z 477.453,A -85,B 0,C 180,E1 -3496.508,E2 -3496.508} C_VEL
LIN {X 0,Y 545.671,Z 488.934,A -85,B 0,C 180,E1 -3497.353,E2 -3497.353} C_VEL
LIN {X 0,Y 545.445,Z 499.655,A -85,B 0,C 180,E1 -3498.309,E2 -3498.309} C_VEL
LIN {X 0,Y 545.247,Z 509.945,A -85,B 0,C 180,E1 -3499.416,E2 -3499.416} C_VEL
LIN {X 0,Y 545.037,Z 518.585,A -85,B 0,C 180,E1 -3500.537,E2 -3500.537} C_VEL
LIN {X 0,Y 544.857,Z 526.872,A -85,B 0,C 180,E1 -3501.843,E2 -3501.843} C_VEL
LIN {X 0,Y 544.737,Z 532.644,A -85,B 0,C 180,E1 -3502.96,E2 -3502.96} C_VEL
LIN {X 0,Y 544.724,Z 538.806,A -85,B 0,C 180,E1 -3504.447,E2 -3504.447} C_VEL
LIN {X 0,Y 544.654,Z 542.318,A -85,B 0,C 180,E1 -3505.56,E2 -3505.56} C_VEL
LIN {X 0,Y 544.647,Z 545.748,A -85,B 0,C 180,E1 -3507.041,E2 -3507.041} C_VEL
LIN {X 0,Y 544.544,Z 547.789,A -85,B 0,C 180,E1 -3508.521,E2 -3508.521} C_VEL
LIN {X 0,Y 544.54,Z 548.496,A -85,B 0,C 180,E1 -3510,E2 -3510} C_VEL
LIN {X 0,Y 544.542,Z 547.878,A -85,B 0,C 180,E1 -3511.479,E2 -3511.479} C_VEL
LIN {X 0,Y 544.646,Z 545.92,A -85,B 0,C 180,E1 -3512.959,E2 -3512.959} C_VEL
LIN {X 0,Y 544.655,Z 542.573,A -85,B 0,C 180,E1 -3514.44,E2 -3514.44} C_VEL
LIN {X 0,Y 544.73,Z 537.742,A -85,B 0,C 180,E1 -3515.924,E2 -3515.924} C_VEL
LIN {X 0,Y 544.783,Z 531.274,A -85,B 0,C 180,E1 -3517.412,E2 -3517.412} C_VEL
LIN {X 0,Y 544.91,Z 524.072,A -85,B 0,C 180,E1 -3518.716,E2 -3518.716} C_VEL
LIN {X 0,Y 545.04,Z 516.529,A -85,B 0,C 180,E1 -3519.837,E2 -3519.837} C_VEL
LIN {X 0,Y 545.276,Z 507.471,A -85,B 0,C 180,E1 -3520.959,E2 -3520.959} C_VEL
LIN {X 0,Y 545.504,Z 496.504,A -85,B 0,C 180,E1 -3522.084,E2 -3522.084} C_VEL
LIN {X 0,Y 545.77,Z 485.346,A -85,B 0,C 180,E1 -3523.023,E2 -3523.023} C_VEL
LIN {X 0,Y 546.083,Z 473.002,A -85,B 0,C 180,E1 -3523.869,E2 -3523.869} C_VEL
LIN {X 0,Y 546.35,Z 461.126,A -85,B 0,C 180,E1 -3524.527,E2 -3524.527} C_VEL
LIN {X 0,Y 546.63,Z 448.71,A -85,B 0,C 180,E1 -3525.07,E2 -3525.07} C_VEL
LIN {X 0,Y 546.78,Z 434.477,A -85,B 0,C 180,E1 -3525.532,E2 -3525.532} C_VEL
LIN {X 0,Y 546.962,Z 419.54,A -85,B 0,C 180,E1 -3525.845,E2 -3525.845} C_VEL
LIN {X 0,Y 547.453,Z 295.752,A -85,B 0,C 180,E1 -3527.498,E2 -3527.498} C_VEL
LIN {X 0,Y 545.759,Z 286.656,A -85,B 0,C 180,E1 -3527.697,E2 -3527.697} C_VEL
LIN {X 0,Y 545.808,Z 279.299,A -85,B 0,C 180,E1 -3528.778,E2 -3528.778} C_VEL
LIN {X 0,Y 546.257,Z 260.26,A -85,B 0,C 180,E1 -3531.708,E2 -3531.708} C_VEL
LIN {X 0,Y 546.233,Z 256.065,A -85,B 0,C 180,E1 -3532.367,E2 -3532.367} C_VEL
LIN {X 0,Y 545.079,Z 250.321,A -85,B 0,C 180,E1 -3533.357,E2 -3533.357} C_VEL
LIN {X 0,Y 545.08,Z 250.215,A -85,B 0,C 180,E1 -3536,E2 -3536} C_VEL
LIN {X 0,Y 545.089,Z 250.203,A -85,B 0,C 180,E1 -3538.748,E2 -3538.748} C_VEL
LIN {X 0,Y 545.058,Z 250.217,A -85,B 0,C 180,E1 -3541.678,E2 -3541.678} C_VEL
LIN {X 0,Y 545.075,Z 250.207,A -85,B 0,C 180,E1 -3544.563,E2 -3544.563} C_VEL
LIN {X 0,Y 545.036,Z 250.22,A -85,B 0,C 180,E1 -3547.303,E2 -3547.303} C_VEL
LIN {X 0,Y 545.068,Z 250.211,A -85,B 0,C 180,E1 -3550.141,E2 -3550.141} C_VEL
LIN {X 0,Y 545.083,Z 250.206,A -85,B 0,C 180,E1 -3553.105,E2 -3553.105} C_VEL
LIN {X 0,Y 545.062,Z 250.209,A -85,B 0,C 180,E1 -3556.223,E2 -3556.223} C_VEL
LIN {X 0,Y 545.095,Z 250.202,A -85,B 0,C 180,E1 -3558.886,E2 -3558.886} C_VEL
LIN {X 0,Y 545.048,Z 250.215,A -85,B 0,C 180,E1 -3561.762,E2 -3561.762} C_VEL
LIN {X 0,Y 545.06,Z 250.21,A -85,B 0,C 180,E1 -3564.533,E2 -3564.533} C_VEL
LIN {X 0,Y 545.075,Z 250.207,A -85,B 0,C 180,E1 -3567.212,E2 -3567.212} C_VEL
LIN {X 0,Y 545.095,Z 250.206,A -85,B 0,C 180,E1 -3569.812,E2 -3569.812} C_VEL
LIN {X 0,Y 545.089,Z 250.213,A -85,B 0,C 180,E1 -3572.825,E2 -3572.825} C_VEL
LIN {X 0,Y 545.045,Z 250.213,A -85,B 0,C 180,E1 -3575.63,E2 -3575.63} C_VEL
LIN {X 0,Y 545.058,Z 250.216,A -85,B 0,C 180,E1 -3578.836,E2 -3578.836} C_VEL
LIN {X 0,Y 545.076,Z 250.213,A -85,B 0,C 180,E1 -3581.195,E2 -3581.195} C_VEL
LIN {X 0,Y 545.069,Z 250.208,A -85,B 0,C 180,E1 -3583.521,E2 -3583.521} C_VEL
LIN {X 0,Y 545.088,Z 250.204,A -85,B 0,C 180,E1 -3585.82,E2 -3585.82} C_VEL
LIN {X 0,Y 545.123,Z 250.209,A -85,B 0,C 180,E1 -3588.849,E2 -3588.849} C_VEL
LIN {X 0,Y 545.122,Z 250.199,A -85,B 0,C 180,E1 -3591.847,E2 -3591.847} C_VEL
LIN {X 0,Y 545.2,Z 250.198,A -85,B 0,C 180,E1 -3594.823,E2 -3594.823} C_VEL
LIN {X 0,Y 545.186,Z 250.19,A -85,B 0,C 180,E1 -3597.784,E2 -3597.784} C_VEL
LIN {X 0,Y 545.208,Z 250.197,A -85,B 0,C 180,E1 -3600.739,E2 -3600.739} C_VEL
LIN {X 0,Y 545.168,Z 250.196,A -85,B 0,C 180,E1 -3602.956,E2 -3602.956} C_VEL
LIN {X 0,Y 545.164,Z 250.198,A -85,B 0,C 180,E1 -3605.92,E2 -3605.92} C_VEL
LIN {X 0,Y 545.119,Z 250.202,A -85,B 0,C 180,E1 -3608.9,E2 -3608.9} C_VEL
LIN {X 0,Y 545.126,Z 250.203,A -85,B 0,C 180,E1 -3611.904,E2 -3611.904} C_VEL
LIN {X 0,Y 545.076,Z 250.207,A -85,B 0,C 180,E1 -3614.944,E2 -3614.944} C_VEL
LIN {X 0,Y 545.074,Z 250.213,A -85,B 0,C 180,E1 -3618.026,E2 -3618.026} C_VEL
LIN {X 0,Y 545.087,Z 250.211,A -85,B 0,C 180,E1 -3620.372,E2 -3620.372} C_VEL
LIN {X 0,Y 545.083,Z 250.208,A -85,B 0,C 180,E1 -3623.559,E2 -3623.559} C_VEL
LIN {X 0,Y 545.072,Z 250.217,A -85,B 0,C 180,E1 -3626.001,E2 -3626.001} C_VEL
LIN {X 0,Y 545.084,Z 250.207,A -85,B 0,C 180,E1 -3628.749,E2 -3628.749} C_VEL
LIN {X 0,Y 545.071,Z 250.214,A -85,B 0,C 180,E1 -3631.683,E2 -3631.683} C_VEL
LIN {X 0,Y 545.075,Z 250.2,A -85,B 0,C 180,E1 -3634.564,E2 -3634.564} C_VEL
LIN {X 0,Y 545.033,Z 250.214,A -85,B 0,C 180,E1 -3637.304,E2 -3637.304} C_VEL
LIN {X 0,Y 545.069,Z 250.211,A -85,B 0,C 180,E1 -3640.142,E2 -3640.142} C_VEL
LIN {X 0,Y 545.073,Z 250.21,A -85,B 0,C 180,E1 -3643.107,E2 -3643.107} C_VEL
LIN {X 0,Y 545.062,Z 250.211,A -85,B 0,C 180,E1 -3646.225,E2 -3646.225} C_VEL
LIN {X 0,Y 545.098,Z 250.201,A -85,B 0,C 180,E1 -3648.888,E2 -3648.888} C_VEL
LIN {X 0,Y 545.05,Z 250.215,A -85,B 0,C 180,E1 -3651.764,E2 -3651.764} C_VEL
LIN {X 0,Y 545.035,Z 250.214,A -85,B 0,C 180,E1 -3654.532,E2 -3654.532} C_VEL
LIN {X 0,Y 545.08,Z 250.211,A -85,B 0,C 180,E1 -3657.213,E2 -3657.213} C_VEL
LIN {X 0,Y 545.064,Z 250.203,A -85,B 0,C 180,E1 -3659.811,E2 -3659.811} C_VEL
LIN {X 0,Y 545.088,Z 250.209,A -85,B 0,C 180,E1 -3662.345,E2 -3662.345} C_VEL
LIN {X 0,Y 545.115,Z 250.271,A -85,B 0,C 180,E1 -3665.584,E2 -3665.584} C_VEL
LIN {X 0,Y 545.3,Z 251.292,A -85,B 0,C 180,E1 -3665.802,E2 -3665.802} C_VEL
LIN {X 0,Y 546.517,Z 258.325,A -85,B 0,C 180,E1 -3666.908,E2 -3666.908} C_VEL
LIN {X 0,Y 546.023,Z 280.198,A -85,B 0,C 180,E1 -3670.103,E2 -3670.103} C_VEL
LIN {X 0,Y 545.753,Z 295.871,A -85,B 0,C 180,E1 -3672.333,E2 -3672.333} C_VEL
LIN {X 0,Y 547.359,Z 304.648,A -85,B 0,C 180,E1 -3672.531,E2 -3672.531} C_VEL
LIN {X 0,Y 546.937,Z 432.596,A -85,B 0,C 180,E1 -3674.25,E2 -3674.25} C_VEL
LIN {X 0,Y 546.771,Z 446.979,A -85,B 0,C 180,E1 -3674.585,E2 -3674.585} C_VEL
LIN {X 0,Y 546.584,Z 460.644,A -85,B 0,C 180,E1 -3675.055,E2 -3675.055} C_VEL
LIN {X 0,Y 546.285,Z 473.845,A -85,B 0,C 180,E1 -3675.662,E2 -3675.662} C_VEL
LIN {X 0,Y 545.939,Z 486.656,A -85,B 0,C 180,E1 -3676.412,E2 -3676.412} C_VEL
LIN {X 0,Y 545.666,Z 498.304,A -85,B 0,C 180,E1 -3677.258,E2 -3677.258} C_VEL
LIN {X 0,Y 545.454,Z 509.087,A -85,B 0,C 180,E1 -3678.209,E2 -3678.209} C_VEL
LIN {X 0,Y 545.231,Z 518.708,A -85,B 0,C 180,E1 -3679.228,E2 -3679.228} C_VEL
LIN {X 0,Y 545.025,Z 527.558,A -85,B 0,C 180,E1 -3680.35,E2 -3680.35} C_VEL
LIN {X 0,Y 544.872,Z 536.035,A -85,B 0,C 180,E1 -3681.657,E2 -3681.657} C_VEL
LIN {X 0,Y 544.736,Z 542.864,A -85,B 0,C 180,E1 -3682.96,E2 -3682.96} C_VEL
LIN {X 0,Y 544.731,Z 547.57,A -85,B 0,C 180,E1 -3684.076,E2 -3684.076} C_VEL
LIN {X 0,Y 544.654,Z 552.444,A -85,B 0,C 180,E1 -3685.56,E2 -3685.56} C_VEL
LIN {X 0,Y 544.646,Z 555.833,A -85,B 0,C 180,E1 -3687.041,E2 -3687.041} C_VEL
LIN {X 0,Y 544.541,Z 557.835,A -85,B 0,C 180,E1 -3688.521,E2 -3688.521} C_VEL
LIN {X 0,Y 544.539,Z 558.5,A -85,B 0,C 180,E1 -3690,E2 -3690} C_VEL
LIN {X 0,Y 544.541,Z 557.836,A -85,B 0,C 180,E1 -3691.479,E2 -3691.479} C_VEL
LIN {X 0,Y 544.646,Z 555.836,A -85,B 0,C 180,E1 -3692.959,E2 -3692.959} C_VEL
LIN {X 0,Y 544.654,Z 552.447,A -85,B 0,C 180,E1 -3694.44,E2 -3694.44} C_VEL
LIN {X 0,Y 544.736,Z 547.568,A -85,B 0,C 180,E1 -3695.924,E2 -3695.924} C_VEL
LIN {X 0,Y 544.783,Z 541.054,A -85,B 0,C 180,E1 -3697.412,E2 -3697.412} C_VEL
LIN {X 0,Y 544.911,Z 533.804,A -85,B 0,C 180,E1 -3698.716,E2 -3698.716} C_VEL
LIN {X 0,Y 545.081,Z 524.823,A -85,B 0,C 180,E1 -3700.024,E2 -3700.024} C_VEL
LIN {X 0,Y 545.35,Z 515.394,A -85,B 0,C 180,E1 -3701.146,E2 -3701.146} C_VEL
LIN {X 0,Y 545.545,Z 504.953,A -85,B 0,C 180,E1 -3702.178,E2 -3702.178} C_VEL
LIN {X 0,Y 545.795,Z 493.417,A -85,B 0,C 180,E1 -3703.117,E2 -3703.117} C_VEL
LIN {X 0,Y 546.118,Z 480.615,A -85,B 0,C 180,E1 -3703.963,E2 -3703.963} C_VEL
LIN {X 0,Y 546.386,Z 468.11,A -85,B 0,C 180,E1 -3704.621,E2 -3704.621} C_VEL
LIN {X 0,Y 546.646,Z 455.635,A -85,B 0,C 180,E1 -3705.133,E2 -3705.133} C_VEL
LIN {X 0,Y 546.845,Z 441.65,A -85,B 0,C 180,E1 -3705.555,E2 -3705.555} C_VEL
LIN {X 0,Y 546.943,Z 426.56,A -85,B 0,C 180,E1 -3705.846,E2 -3705.846} C_VEL
LIN {X 0,Y 547.363,Z 304.674,A -85,B 0,C 180,E1 -3707.468,E2 -3707.468} C_VEL
LIN {X 0,Y 545.77,Z 296.104,A -85,B 0,C 180,E1 -3707.652,E2 -3707.652} C_VEL
LIN {X 0,Y 545.842,Z 290.664,A -85,B 0,C 180,E1 -3708.388,E2 -3708.388} C_VEL
LIN {X 0,Y 546.214,Z 270.454,A -85,B 0,C 180,E1 -3711.314,E2 -3711.314} C_VEL
LIN {X 0,Y 546.548,Z 258.325,A -85,B 0,C 180,E1 -3713.091,E2 -3713.091} C_VEL
LIN {X 0,Y 545.146,Z 250.562,A -85,B 0,C 180,E1 -3714.328,E2 -3714.328} C_VEL
LIN {X 0,Y 545.099,Z 250.212,A -85,B 0,C 180,E1 -3714.569,E2 -3714.569} C_VEL
LIN {X 0,Y 545.088,Z 250.209,A -85,B 0,C 180,E1 -3717.655,E2 -3717.655} C_VEL
LIN {X 0,Y 545.076,Z 250.202,A -85,B 0,C 180,E1 -3720.246,E2 -3720.246} C_VEL
LIN {X 0,Y 545.087,Z 250.207,A -85,B 0,C 180,E1 -3723.063,E2 -3723.063} C_VEL
LIN {X 0,Y 545.031,Z 250.215,A -85,B 0,C 180,E1 -3725.672,E2 -3725.672} C_VEL
LIN {X 0,Y 545.049,Z 250.215,A -85,B 0,C 180,E1 -3728.237,E2 -3728.237} C_VEL
LIN {X 0,Y 545.084,Z 250.203,A -85,B 0,C 180,E1 -3731.113,E2 -3731.113} C_VEL
LIN {X 0,Y 545.055,Z 250.216,A -85,B 0,C 180,E1 -3734.128,E2 -3734.128} C_VEL
LIN {X 0,Y 545.074,Z 250.21,A -85,B 0,C 180,E1 -3736.893,E2 -3736.893} C_VEL
LIN {X 0,Y 545.07,Z 250.211,A -85,B 0,C 180,E1 -3739.858,E2 -3739.858} C_VEL
LIN {X 0,Y 545.069,Z 250.207,A -85,B 0,C 180,E1 -3743.073,E2 -3743.073} C_VEL
LIN {X 0,Y 545.08,Z 250.2,A -85,B 0,C 180,E1 -3745.606,E2 -3745.606} C_VEL
LIN {X 0,Y 545.072,Z 250.214,A -85,B 0,C 180,E1 -3748.317,E2 -3748.317} C_VEL
LIN {X 0,Y 545.085,Z 250.207,A -85,B 0,C 180,E1 -3751.251,E2 -3751.251} C_VEL
LIN {X 0,Y 545.082,Z 250.215,A -85,B 0,C 180,E1 -3754,E2 -3754} C_VEL
LIN {X 0,Y 545.084,Z 250.208,A -85,B 0,C 180,E1 -3756.441,E2 -3756.441} C_VEL
LIN {X 0,Y 545.087,Z 250.211,A -85,B 0,C 180,E1 -3759.628,E2 -3759.628} C_VEL
LIN {X 0,Y 545.087,Z 250.204,A -85,B 0,C 180,E1 -3762.75,E2 -3762.75} C_VEL
LIN {X 0,Y 545.088,Z 250.215,A -85,B 0,C 180,E1 -3765.82,E2 -3765.82} C_VEL
LIN {X 0,Y 545.109,Z 250.202,A -85,B 0,C 180,E1 -3768.849,E2 -3768.849} C_VEL
LIN {X 0,Y 545.123,Z 250.208,A -85,B 0,C 180,E1 -3771.847,E2 -3771.847} C_VEL
LIN {X 0,Y 545.199,Z 250.191,A -85,B 0,C 180,E1 -3774.823,E2 -3774.823} C_VEL
LIN {X 0,Y 545.187,Z 250.2,A -85,B 0,C 180,E1 -3777.784,E2 -3777.784} C_VEL
LIN {X 0,Y 545.207,Z 250.191,A -85,B 0,C 180,E1 -3780.739,E2 -3780.739} C_VEL
LIN {X 0,Y 545.168,Z 250.194,A -85,B 0,C 180,E1 -3782.956,E2 -3782.956} C_VEL
LIN {X 0,Y 545.164,Z 250.199,A -85,B 0,C 180,E1 -3785.92,E2 -3785.92} C_VEL
LIN {X 0,Y 545.114,Z 250.203,A -85,B 0,C 180,E1 -3788.9,E2 -3788.9} C_VEL
LIN {X 0,Y 545.127,Z 250.203,A -85,B 0,C 180,E1 -3791.904,E2 -3791.904} C_VEL
LIN {X 0,Y 545.078,Z 250.21,A -85,B 0,C 180,E1 -3794.944,E2 -3794.944} C_VEL
LIN {X 0,Y 545.075,Z 250.208,A -85,B 0,C 180,E1 -3798.026,E2 -3798.026} C_VEL
LIN {X 0,Y 545.088,Z 250.205,A -85,B 0,C 180,E1 -3800.372,E2 -3800.372} C_VEL
LIN {X 0,Y 545.084,Z 250.21,A -85,B 0,C 180,E1 -3803.559,E2 -3803.559} C_VEL
LIN {X 0,Y 545.073,Z 250.205,A -85,B 0,C 180,E1 -3806.001,E2 -3806.001} C_VEL
LIN {X 0,Y 545.086,Z 250.212,A -85,B 0,C 180,E1 -3808.749,E2 -3808.749} C_VEL
LIN {X 0,Y 545.072,Z 250.204,A -85,B 0,C 180,E1 -3811.683,E2 -3811.683} C_VEL
LIN {X 0,Y 545.076,Z 250.203,A -85,B 0,C 180,E1 -3814.564,E2 -3814.564} C_VEL
LIN {X 0,Y 545.06,Z 250.217,A -85,B 0,C 180,E1 -3817.015,E2 -3817.015} C_VEL
LIN {X 0,Y 544.351,Z 250.301,A -85,B 0,C 180,E1 -3817.632,E2 -3817.632} C_VEL
LIN {X 0,Y 541.484,Z 250.663,A -85,B 0,C 180,E1 -3818.633,E2 -3818.633} C_VEL
LIN {X 0,Y 539.101,Z 250.953,A -85,B 0,C 180,E1 -3819.438,E2 -3819.438} C_VEL
LIN {X 0,Y 538.101,Z 251.075,A -85,B 0,C 180,E1 -3820.06,E2 -3820.06} C_VEL
LIN {X 0,Y 538.03,Z 251.082,A -85,B 0,C 180,E1 -3820.271,E2 -3820.271} C_VEL
LIN {X 0,Y 538.022,Z 251.091,A -85,B 0,C 180,E1 -3822.988,E2 -3822.988} C_VEL
LIN {X 0,Y 538.026,Z 251.087,A -85,B 0,C 180,E1 -3825.926,E2 -3825.926} C_VEL
LIN {X 0,Y 538.049,Z 251.085,A -85,B 0,C 180,E1 -3829.225,E2 -3829.225} C_VEL
LIN {X 0,Y 537.991,Z 251.092,A -85,B 0,C 180,E1 -3832.123,E2 -3832.123} C_VEL
LIN {X 0,Y 538.011,Z 251.09,A -85,B 0,C 180,E1 -3834.917,E2 -3834.917} C_VEL
LIN {X 0,Y 538.026,Z 251.088,A -85,B 0,C 180,E1 -3837.619,E2 -3837.619} C_VEL
LIN {X 0,Y 538.017,Z 251.096,A -85,B 0,C 180,E1 -3840.239,E2 -3840.239} C_VEL
LIN {X 0,Y 538.064,Z 251.086,A -85,B 0,C 180,E1 -3842.797,E2 -3842.797} C_VEL
LIN {X 0,Y 538.029,Z 251.083,A -85,B 0,C 180,E1 -3845.292,E2 -3845.292} C_VEL
LIN {X 0,Y 538.082,Z 251.306,A -85,B 0,C 180,E1 -3846.575,E2 -3846.575} C_VEL
LIN {X 0,Y 539.409,Z 258.473,A -85,B 0,C 180,E1 -3847.8,E2 -3847.8} C_VEL
LIN {X 0,Y 538.926,Z 277.497,A -85,B 0,C 180,E1 -3850.775,E2 -3850.775} C_VEL
LIN {X 0,Y 538.798,Z 286.595,A -85,B 0,C 180,E1 -3852.149,E2 -3852.149} C_VEL
LIN {X 0,Y 540.413,Z 295.165,A -85,B 0,C 180,E1 -3852.348,E2 -3852.348} C_VEL
LIN {X 0,Y 540.695,Z 300.122,A -85,B 0,C 180,E1 -3852.425,E2 -3852.425} C_VEL
LIN {X 0,Y 540.131,Z 422.983,A -85,B 0,C 180,E1 -3854.094,E2 -3854.094} C_VEL
LIN {X 0,Y 539.891,Z 437.691,A -85,B 0,C 180,E1 -3854.445,E2 -3854.445} C_VEL
LIN {X 0,Y 539.639,Z 451.895,A -85,B 0,C 180,E1 -3854.951,E2 -3854.951} C_VEL
LIN {X 0,Y 539.371,Z 464.923,A -85,B 0,C 180,E1 -3855.57,E2 -3855.57} C_VEL
LIN {X 0,Y 539.023,Z 477.529,A -85,B 0,C 180,E1 -3856.331,E2 -3856.331} C_VEL
LIN {X 0,Y 538.74,Z 489.008,A -85,B 0,C 180,E1 -3857.187,E2 -3857.187} C_VEL
LIN {X 0,Y 538.461,Z 500.282,A -85,B 0,C 180,E1 -3858.21,E2 -3858.21} C_VEL
LIN {X 0,Y 538.236,Z 509.996,A -85,B 0,C 180,E1 -3859.277,E2 -3859.277} C_VEL
LIN {X 0,Y 537.973,Z 518.62,A -85,B 0,C 180,E1 -3860.412,E2 -3860.412} C_VEL
LIN {X 0,Y 537.809,Z 526.889,A -85,B 0,C 180,E1 -3861.735,E2 -3861.735} C_VEL
LIN {X 0,Y 537.662,Z 532.649,A -85,B 0,C 180,E1 -3862.867,E2 -3862.867} C_VEL
LIN {X 0,Y 537.655,Z 538.808,A -85,B 0,C 180,E1 -3864.374,E2 -3864.374} C_VEL
LIN {X 0,Y 537.55,Z 542.319,A -85,B 0,C 180,E1 -3865.501,E2 -3865.501} C_VEL
LIN {X 0,Y 537.547,Z 545.749,A -85,B 0,C 180,E1 -3867.002,E2 -3867.002} C_VEL
LIN {X 0,Y 537.45,Z 547.79,A -85,B 0,C 180,E1 -3868.501,E2 -3868.501} C_VEL
LIN {X 0,Y 537.441,Z 548.496,A -85,B 0,C 180,E1 -3870,E2 -3870} C_VEL
LIN {X 0,Y 537.448,Z 547.878,A -85,B 0,C 180,E1 -3871.499,E2 -3871.499} C_VEL
LIN {X 0,Y 537.546,Z 545.919,A -85,B 0,C 180,E1 -3872.998,E2 -3872.998} C_VEL
LIN {X 0,Y 537.551,Z 542.571,A -85,B 0,C 180,E1 -3874.499,E2 -3874.499} C_VEL
LIN {X 0,Y 537.643,Z 537.74,A -85,B 0,C 180,E1 -3876.002,E2 -3876.002} C_VEL
LIN {X 0,Y 537.661,Z 533.081,A -85,B 0,C 180,E1 -3877.133,E2 -3877.133} C_VEL
LIN {X 0,Y 537.824,Z 526.315,A -85,B 0,C 180,E1 -3878.453,E2 -3878.453} C_VEL
LIN {X 0,Y 537.952,Z 517.911,A -85,B 0,C 180,E1 -3879.778,E2 -3879.778} C_VEL
LIN {X 0,Y 538.217,Z 509.141,A -85,B 0,C 180,E1 -3880.914,E2 -3880.914} C_VEL
LIN {X 0,Y 538.466,Z 498.513,A -85,B 0,C 180,E1 -3882.053,E2 -3882.053} C_VEL
LIN {X 0,Y 538.768,Z 487.767,A -85,B 0,C 180,E1 -3883.004,E2 -3883.004} C_VEL
LIN {X 0,Y 539.104,Z 476.012,A -85,B 0,C 180,E1 -3883.859,E2 -3883.859} C_VEL
LIN {X 0,Y 539.446,Z 463.045,A -85,B 0,C 180,E1 -3884.62,E2 -3884.62} C_VEL
LIN {X 0,Y 539.715,Z 451.103,A -85,B 0,C 180,E1 -3885.172,E2 -3885.172} C_VEL
LIN {X 0,Y 539.914,Z 437.28,A -85,B 0,C 180,E1 -3885.657,E2 -3885.657} C_VEL
LIN {X 0,Y 540.106,Z 422.578,A -85,B 0,C 180,E1 -3886.003,E2 -3886.003} C_VEL
LIN {X 0,Y 540.643,Z 296.297,A -85,B 0,C 180,E1 -3887.719,E2 -3887.719} C_VEL
LIN {X 0,Y 538.803,Z 286.736,A -85,B 0,C 180,E1 -3887.931,E2 -3887.931} C_VEL
LIN {X 0,Y 538.89,Z 279.354,A -85,B 0,C 180,E1 -3889.028,E2 -3889.028} C_VEL
LIN {X 0,Y 539.417,Z 259.041,A -85,B 0,C 180,E1 -3892.199,E2 -3892.199} C_VEL
LIN {X 0,Y 538.357,Z 252.704,A -85,B 0,C 180,E1 -3893.259,E2 -3893.259} C_VEL
LIN {X 0,Y 538.049,Z 251.135,A -85,B 0,C 180,E1 -3893.577,E2 -3893.577} C_VEL
LIN {X 0,Y 538.042,Z 251.089,A -85,B 0,C 180,E1 -3896.366,E2 -3896.366} C_VEL
LIN {X 0,Y 538.03,Z 251.083,A -85,B 0,C 180,E1 -3898.933,E2 -3898.933} C_VEL
LIN {X 0,Y 538.013,Z 251.095,A -85,B 0,C 180,E1 -3901.887,E2 -3901.887} C_VEL
LIN {X 0,Y 538.024,Z 251.086,A -85,B 0,C 180,E1 -3904.619,E2 -3904.619} C_VEL
LIN {X 0,Y 538.004,Z 251.094,A -85,B 0,C 180,E1 -3907.17,E2 -3907.17} C_VEL
LIN {X 0,Y 538.024,Z 251.092,A -85,B 0,C 180,E1 -3909.796,E2 -3909.796} C_VEL
LIN {X 0,Y 538.02,Z 251.082,A -85,B 0,C 180,E1 -3912.785,E2 -3912.785} C_VEL
LIN {X 0,Y 538.025,Z 251.088,A -85,B 0,C 180,E1 -3915.925,E2 -3915.925} C_VEL
LIN {X 0,Y 538.073,Z 251.079,A -85,B 0,C 180,E1 -3919.248,E2 -3919.248} C_VEL
LIN {X 0,Y 537.988,Z 251.092,A -85,B 0,C 180,E1 -3922.122,E2 -3922.122} C_VEL
LIN {X 0,Y 538.015,Z 251.091,A -85,B 0,C 180,E1 -3924.917,E2 -3924.917} C_VEL
LIN {X 0,Y 538.025,Z 251.084,A -85,B 0,C 180,E1 -3927.618,E2 -3927.618} C_VEL
LIN {X 0,Y 538.036,Z 251.085,A -85,B 0,C 180,E1 -3930.24,E2 -3930.24} C_VEL
LIN {X 0,Y 538.059,Z 251.088,A -85,B 0,C 180,E1 -3932.796,E2 -3932.796} C_VEL
LIN {X 0,Y 538.041,Z 251.089,A -85,B 0,C 180,E1 -3935.292,E2 -3935.292} C_VEL
LIN {X 0,Y 538.007,Z 251.088,A -85,B 0,C 180,E1 -3938.041,E2 -3938.041} C_VEL
LIN {X 0,Y 538.032,Z 251.094,A -85,B 0,C 180,E1 -3940.94,E2 -3940.94} C_VEL
LIN {X 0,Y 538.019,Z 251.088,A -85,B 0,C 180,E1 -3943.299,E2 -3943.299} C_VEL
LIN {X 0,Y 538.056,Z 251.08,A -85,B 0,C 180,E1 -3945.63,E2 -3945.63} C_VEL
LIN {X 0,Y 538.081,Z 251.088,A -85,B 0,C 180,E1 -3948.702,E2 -3948.702} C_VEL
LIN {X 0,Y 538.079,Z 251.076,A -85,B 0,C 180,E1 -3951.739,E2 -3951.739} C_VEL
LIN {X 0,Y 538.176,Z 251.074,A -85,B 0,C 180,E1 -3954.755,E2 -3954.755} C_VEL
LIN {X 0,Y 538.158,Z 251.065,A -85,B 0,C 180,E1 -3957.755,E2 -3957.755} C_VEL
LIN {X 0,Y 538.177,Z 251.073,A -85,B 0,C 180,E1 -3960.748,E2 -3960.748} C_VEL
LIN {X 0,Y 538.134,Z 251.071,A -85,B 0,C 180,E1 -3962.994,E2 -3962.994} C_VEL
LIN {X 0,Y 538.116,Z 251.076,A -85,B 0,C 180,E1 -3965.997,E2 -3965.997} C_VEL
LIN {X 0,Y 538.068,Z 251.08,A -85,B 0,C 180,E1 -3969.018,E2 -3969.018} C_VEL
LIN {X 0,Y 538.074,Z 251.083,A -85,B 0,C 180,E1 -3972.063,E2 -3972.063} C_VEL
LIN {X 0,Y 538.037,Z 251.083,A -85,B 0,C 180,E1 -3975.144,E2 -3975.144} C_VEL
LIN {X 0,Y 538.026,Z 251.095,A -85,B 0,C 180,E1 -3978.27,E2 -3978.27} C_VEL
LIN {X 0,Y 538.031,Z 251.086,A -85,B 0,C 180,E1 -3980.652,E2 -3980.652} C_VEL
LIN {X 0,Y 538.016,Z 251.092,A -85,B 0,C 180,E1 -3983.888,E2 -3983.888} C_VEL
LIN {X 0,Y 538.035,Z 251.087,A -85,B 0,C 180,E1 -3986.367,E2 -3986.367} C_VEL
LIN {X 0,Y 538.049,Z 251.083,A -85,B 0,C 180,E1 -3988.939,E2 -3988.939} C_VEL
LIN {X 0,Y 538.021,Z 251.092,A -85,B 0,C 180,E1 -3991.891,E2 -3991.891} C_VEL
LIN {X 0,Y 538.025,Z 251.077,A -85,B 0,C 180,E1 -3994.621,E2 -3994.621} C_VEL
LIN {X 0,Y 538.002,Z 251.088,A -85,B 0,C 180,E1 -3997.171,E2 -3997.171} C_VEL
LIN {X 0,Y 538.025,Z 251.093,A -85,B 0,C 180,E1 -3999.797,E2 -3999.797} C_VEL
LIN {X 0,Y 538.014,Z 251.088,A -85,B 0,C 180,E1 -4002.787,E2 -4002.787} C_VEL
LIN {X 0,Y 538.025,Z 251.091,A -85,B 0,C 180,E1 -4005.926,E2 -4005.926} C_VEL
LIN {X 0,Y 538.075,Z 251.079,A -85,B 0,C 180,E1 -4009.25,E2 -4009.25} C_VEL
LIN {X 0,Y 537.989,Z 251.09,A -85,B 0,C 180,E1 -4012.123,E2 -4012.123} C_VEL
LIN {X 0,Y 537.997,Z 251.093,A -85,B 0,C 180,E1 -4014.916,E2 -4014.916} C_VEL
LIN {X 0,Y 538.025,Z 251.094,A -85,B 0,C 180,E1 -4017.619,E2 -4017.619} C_VEL
LIN {X 0,Y 538.016,Z 251.078,A -85,B 0,C 180,E1 -4020.24,E2 -4020.24} C_VEL
LIN {X 0,Y 538.062,Z 251.087,A -85,B 0,C 180,E1 -4022.797,E2 -4022.797} C_VEL
LIN {X 0,Y 538.084,Z 251.156,A -85,B 0,C 180,E1 -4025.39,E2 -4025.39} C_VEL
LIN {X 0,Y 538.362,Z 252.67,A -85,B 0,C 180,E1 -4025.689,E2 -4025.689} C_VEL
LIN {X 0,Y 539.625,Z 259.617,A -85,B 0,C 180,E1 -4026.799,E2 -4026.799} C_VEL
LIN {X 0,Y 539.107,Z 280.837,A -85,B 0,C 180,E1 -4029.94,E2 -4029.94} C_VEL
LIN {X 0,Y 538.793,Z 295.944,A -85,B 0,C 180,E1 -4032.107,E2 -4032.107} C_VEL
LIN {X 0,Y 540.701,Z 307.108,A -85,B 0,C 180,E1 -4032.344,E2 -4032.344} C_VEL
LIN {X 0,Y 540.103,Z 433.777,A -85,B 0,C 180,E1 -4034.069,E2 -4034.069} C_VEL
LIN {X 0,Y 539.892,Z 448.301,A -85,B 0,C 180,E1 -4034.427,E2 -4034.427} C_VEL
LIN {X 0,Y 539.589,Z 462.732,A -85,B 0,C 180,E1 -4034.949,E2 -4034.949} C_VEL
LIN {X 0,Y 539.373,Z 475.545,A -85,B 0,C 180,E1 -4035.57,E2 -4035.57} C_VEL
LIN {X 0,Y 538.985,Z 488.016,A -85,B 0,C 180,E1 -4036.33,E2 -4036.33} C_VEL
LIN {X 0,Y 538.675,Z 500.585,A -85,B 0,C 180,E1 -4037.282,E2 -4037.282} C_VEL
LIN {X 0,Y 538.433,Z 510.772,A -85,B 0,C 180,E1 -4038.224,E2 -4038.224} C_VEL
LIN {X 0,Y 538.186,Z 520.298,A -85,B 0,C 180,E1 -4039.276,E2 -4039.276} C_VEL
LIN {X 0,Y 537.969,Z 528.889,A -85,B 0,C 180,E1 -4040.412,E2 -4040.412} C_VEL
LIN {X 0,Y 537.804,Z 537.115,A -85,B 0,C 180,E1 -4041.735,E2 -4041.735} C_VEL
LIN {X 0,Y 537.661,Z 542.864,A -85,B 0,C 180,E1 -4042.867,E2 -4042.867} C_VEL
LIN {X 0,Y 537.655,Z 548.961,A -85,B 0,C 180,E1 -4044.374,E2 -4044.374} C_VEL
LIN {X 0,Y 537.55,Z 552.444,A -85,B 0,C 180,E1 -4045.501,E2 -4045.501} C_VEL
LIN {X 0,Y 537.547,Z 555.832,A -85,B 0,C 180,E1 -4047.002,E2 -4047.002} C_VEL
LIN {X 0,Y 537.447,Z 557.835,A -85,B 0,C 180,E1 -4048.501,E2 -4048.501} C_VEL
LIN {X 0,Y 537.44,Z 558.5,A -85,B 0,C 180,E1 -4050,E2 -4050} C_VEL
LIN {X 0,Y 537.447,Z 557.837,A -85,B 0,C 180,E1 -4051.499,E2 -4051.499} C_VEL
LIN {X 0,Y 537.547,Z 555.836,A -85,B 0,C 180,E1 -4052.998,E2 -4052.998} C_VEL
LIN {X 0,Y 537.55,Z 552.447,A -85,B 0,C 180,E1 -4054.499,E2 -4054.499} C_VEL
LIN {X 0,Y 537.65,Z 547.568,A -85,B 0,C 180,E1 -4056.003,E2 -4056.003} C_VEL
LIN {X 0,Y 537.704,Z 541.054,A -85,B 0,C 180,E1 -4057.51,E2 -4057.51} C_VEL
LIN {X 0,Y 537.86,Z 533.792,A -85,B 0,C 180,E1 -4058.832,E2 -4058.832} C_VEL
LIN {X 0,Y 538.033,Z 524.793,A -85,B 0,C 180,E1 -4060.157,E2 -4060.157} C_VEL
LIN {X 0,Y 538.342,Z 515.348,A -85,B 0,C 180,E1 -4061.293,E2 -4061.293} C_VEL
LIN {X 0,Y 538.548,Z 504.89,A -85,B 0,C 180,E1 -4062.339,E2 -4062.339} C_VEL
LIN {X 0,Y 538.87,Z 493.351,A -85,B 0,C 180,E1 -4063.289,E2 -4063.289} C_VEL
LIN {X 0,Y 539.19,Z 480.548,A -85,B 0,C 180,E1 -4064.146,E2 -4064.146} C_VEL
LIN {X 0,Y 539.508,Z 468.043,A -85,B 0,C 180,E1 -4064.812,E2 -4064.812} C_VEL
LIN {X 0,Y 539.793,Z 454.732,A -85,B 0,C 180,E1 -4065.361,E2 -4065.361} C_VEL
LIN {X 0,Y 540.031,Z 440.669,A -85,B 0,C 180,E1 -4065.781,E2 -4065.781} C_VEL
LIN {X 0,Y 540.112,Z 426.493,A -85,B 0,C 180,E1 -4066.052,E2 -4066.052} C_VEL
LIN {X 0,Y 540.663,Z 306.001,A -85,B 0,C 180,E1 -4067.673,E2 -4067.673} C_VEL
LIN {X 0,Y 538.778,Z 295.865,A -85,B 0,C 180,E1 -4067.899,E2 -4067.899} C_VEL
LIN {X 0,Y 539.195,Z 277.135,A -85,B 0,C 180,E1 -4070.605,E2 -4070.605} C_VEL
LIN {X 0,Y 539.629,Z 259.617,A -85,B 0,C 180,E1 -4073.201,E2 -4073.201} C_VEL
LIN {X 0,Y 538.121,Z 251.483,A -85,B 0,C 180,E1 -4074.513,E2 -4074.513} C_VEL
LIN {X 0,Y 538.077,Z 251.088,A -85,B 0,C 180,E1 -4074.705,E2 -4074.705} C_VEL
LIN {X 0,Y 538.057,Z 251.086,A -85,B 0,C 180,E1 -4077.352,E2 -4077.352} C_VEL
LIN {X 0,Y 538.016,Z 251.078,A -85,B 0,C 180,E1 -4079.761,E2 -4079.761} C_VEL
LIN {X 0,Y 538.025,Z 251.094,A -85,B 0,C 180,E1 -4082.382,E2 -4082.382} C_VEL
LIN {X 0,Y 537.996,Z 251.093,A -85,B 0,C 180,E1 -4085.084,E2 -4085.084} C_VEL
LIN {X 0,Y 537.989,Z 251.09,A -85,B 0,C 180,E1 -4087.877,E2 -4087.877} C_VEL
LIN {X 0,Y 538.045,Z 251.082,A -85,B 0,C 180,E1 -4090.775,E2 -4090.775} C_VEL
LIN {X 0,Y 538.025,Z 251.091,A -85,B 0,C 180,E1 -4094.074,E2 -4094.074} C_VEL
LIN {X 0,Y 538.014,Z 251.088,A -85,B 0,C 180,E1 -4097.213,E2 -4097.213} C_VEL
LIN {X 0,Y 538.025,Z 251.093,A -85,B 0,C 180,E1 -4100.203,E2 -4100.203} C_VEL
LIN {X 0,Y 538.023,Z 251.084,A -85,B 0,C 180,E1 -4103.067,E2 -4103.067} C_VEL
LIN {X 0,Y 538.021,Z 251.081,A -85,B 0,C 180,E1 -4105.827,E2 -4105.827} C_VEL
LIN {X 0,Y 538.018,Z 251.09,A -85,B 0,C 180,E1 -4108.499,E2 -4108.499} C_VEL
LIN {X 0,Y 538.052,Z 251.082,A -85,B 0,C 180,E1 -4111.099,E2 -4111.099} C_VEL
LIN {X 0,Y 538.043,Z 251.086,A -85,B 0,C 180,E1 -4113.633,E2 -4113.633} C_VEL
LIN {X 0,Y 538.015,Z 251.092,A -85,B 0,C 180,E1 -4116.118,E2 -4116.118} C_VEL
LIN {X 0,Y 538.031,Z 251.086,A -85,B 0,C 180,E1 -4119.348,E2 -4119.348} C_VEL
LIN {X 0,Y 538.065,Z 251.08,A -85,B 0,C 180,E1 -4122.517,E2 -4122.517} C_VEL
LIN {X 0,Y 538.056,Z 251.088,A -85,B 0,C 180,E1 -4125.63,E2 -4125.63} C_VEL
LIN {X 0,Y 538.068,Z 251.078,A -85,B 0,C 180,E1 -4128.701,E2 -4128.701} C_VEL
LIN {X 0,Y 538.079,Z 251.088,A -85,B 0,C 180,E1 -4131.74,E2 -4131.74} C_VEL
LIN {X 0,Y 538.156,Z 251.068,A -85,B 0,C 180,E1 -4134.755,E2 -4134.755} C_VEL
LIN {X 0,Y 538.159,Z 251.076,A -85,B 0,C 180,E1 -4137.755,E2 -4137.755} C_VEL
LIN {X 0,Y 538.177,Z 251.067,A -85,B 0,C 180,E1 -4140.748,E2 -4140.748} C_VEL
LIN {X 0,Y 538.134,Z 251.07,A -85,B 0,C 180,E1 -4142.995,E2 -4142.995} C_VEL
LIN {X 0,Y 538.117,Z 251.076,A -85,B 0,C 180,E1 -4145.997,E2 -4145.997} C_VEL
LIN {X 0,Y 538.065,Z 251.082,A -85,B 0,C 180,E1 -4149.018,E2 -4149.018} C_VEL
LIN {X 0,Y 538.075,Z 251.08,A -85,B 0,C 180,E1 -4152.063,E2 -4152.063} C_VEL
LIN {X 0,Y 538.038,Z 251.089,A -85,B 0,C 180,E1 -4155.144,E2 -4155.144} C_VEL
LIN {X 0,Y 538.027,Z 251.086,A -85,B 0,C 180,E1 -4158.27,E2 -4158.27} C_VEL
LIN {X 0,Y 538.032,Z 251.086,A -85,B 0,C 180,E1 -4160.652,E2 -4160.652} C_VEL
LIN {X 0,Y 538.017,Z 251.088,A -85,B 0,C 180,E1 -4163.888,E2 -4163.888} C_VEL
LIN {X 0,Y 538.036,Z 251.083,A -85,B 0,C 180,E1 -4166.367,E2 -4166.367} C_VEL
LIN {X 0,Y 538.05,Z 251.092,A -85,B 0,C 180,E1 -4168.939,E2 -4168.939} C_VEL
LIN {X 0,Y 538.021,Z 251.081,A -85,B 0,C 180,E1 -4171.891,E2 -4171.891} C_VEL
LIN {X 0,Y 538.026,Z 251.081,A -85,B 0,C 180,E1 -4174.621,E2 -4174.621} C_VEL
LIN {X 0,Y 538.003,Z 251.094,A -85,B 0,C 180,E1 -4177.171,E2 -4177.171} C_VEL
LIN {X 0,Y 538.03,Z 251.082,A -85,B 0,C 180,E1 -4180.271,E2 -4180.271} C_VEL
LIN {X 0,Y 537.39,Z 251.165,A -85,B 0,C 180,E1 -4180.896,E2 -4180.896} C_VEL
LIN {X 0,Y 534.535,Z 251.522,A -85,B 0,C 180,E1 -4181.911,E2 -4181.911} C_VEL
LIN {X 0,Y 532.099,Z 251.825,A -85,B 0,C 180,E1 -4182.728,E2 -4182.728} C_VEL
LIN {X 0,Y 531.046,Z 251.956,A -85,B 0,C 180,E1 -4183.359,E2 -4183.359} C_VEL
LIN {X 0,Y 530.958,Z 251.966,A -85,B 0,C 180,E1 -4183.572,E2 -4183.572} C_VEL
LIN {X 0,Y 530.964,Z 251.972,A -85,B 0,C 180,E1 -4186.506,E2 -4186.506} C_VEL
LIN {X 0,Y 530.987,Z 251.967,A -85,B 0,C 180,E1 -4188.976,E2 -4188.976} C_VEL
LIN {X 0,Y 530.955,Z 251.966,A -85,B 0,C 180,E1 -4191.53,E2 -4191.53} C_VEL
LIN {X 0,Y 530.975,Z 251.972,A -85,B 0,C 180,E1 -4194.382,E2 -4194.382} C_VEL
LIN {X 0,Y 530.97,Z 251.968,A -85,B 0,C 180,E1 -4197.134,E2 -4197.134} C_VEL
LIN {X 0,Y 530.969,Z 251.968,A -85,B 0,C 180,E1 -4199.804,E2 -4199.804} C_VEL
LIN {X 0,Y 531.015,Z 251.959,A -85,B 0,C 180,E1 -4202.468,E2 -4202.468} C_VEL
LIN {X 0,Y 530.996,Z 251.959,A -85,B 0,C 180,E1 -4204.943,E2 -4204.943} C_VEL
LIN {X 0,Y 531.034,Z 252.19,A -85,B 0,C 180,E1 -4206.378,E2 -4206.378} C_VEL
LIN {X 0,Y 532.476,Z 259.616,A -85,B 0,C 180,E1 -4207.67,E2 -4207.67} C_VEL
LIN {X 0,Y 532.039,Z 277.565,A -85,B 0,C 180,E1 -4210.517,E2 -4210.517} C_VEL
LIN {X 0,Y 531.848,Z 286.704,A -85,B 0,C 180,E1 -4211.911,E2 -4211.911} C_VEL
LIN {X 0,Y 533.948,Z 298.484,A -85,B 0,C 180,E1 -4212.171,E2 -4212.171} C_VEL
LIN {X 0,Y 533.309,Z 423.084,A -85,B 0,C 180,E1 -4213.885,E2 -4213.885} C_VEL
LIN {X 0,Y 533.052,Z 437.493,A -85,B 0,C 180,E1 -4214.231,E2 -4214.231} C_VEL
LIN {X 0,Y 532.825,Z 450.847,A -85,B 0,C 180,E1 -4214.705,E2 -4214.705} C_VEL
LIN {X 0,Y 532.565,Z 463.236,A -85,B 0,C 180,E1 -4215.284,E2 -4215.284} C_VEL
LIN {X 0,Y 532.149,Z 476.182,A -85,B 0,C 180,E1 -4216.053,E2 -4216.053} C_VEL
LIN {X 0,Y 531.831,Z 487.911,A -85,B 0,C 180,E1 -4216.921,E2 -4216.921} C_VEL
LIN {X 0,Y 531.469,Z 499.353,A -85,B 0,C 180,E1 -4217.953,E2 -4217.953} C_VEL
LIN {X 0,Y 531.222,Z 510.068,A -85,B 0,C 180,E1 -4219.133,E2 -4219.133} C_VEL
LIN {X 0,Y 530.93,Z 518.691,A -85,B 0,C 180,E1 -4220.284,E2 -4220.284} C_VEL
LIN {X 0,Y 530.742,Z 526.96,A -85,B 0,C 180,E1 -4221.625,E2 -4221.625} C_VEL
LIN {X 0,Y 530.587,Z 532.718,A -85,B 0,C 180,E1 -4222.771,E2 -4222.771} C_VEL
LIN {X 0,Y 530.585,Z 538.864,A -85,B 0,C 180,E1 -4224.299,E2 -4224.299} C_VEL
LIN {X 0,Y 530.45,Z 542.367,A -85,B 0,C 180,E1 -4225.441,E2 -4225.441} C_VEL
LIN {X 0,Y 530.453,Z 545.787,A -85,B 0,C 180,E1 -4226.962,E2 -4226.962} C_VEL
LIN {X 0,Y 530.36,Z 547.823,A -85,B 0,C 180,E1 -4228.481,E2 -4228.481} C_VEL
LIN {X 0,Y 530.342,Z 548.528,A -85,B 0,C 180,E1 -4230,E2 -4230} C_VEL
LIN {X 0,Y 530.358,Z 547.91,A -85,B 0,C 180,E1 -4231.519,E2 -4231.519} C_VEL
LIN {X 0,Y 530.452,Z 545.955,A -85,B 0,C 180,E1 -4233.038,E2 -4233.038} C_VEL
LIN {X 0,Y 530.45,Z 542.615,A -85,B 0,C 180,E1 -4234.559,E2 -4234.559} C_VEL
LIN {X 0,Y 530.556,Z 537.794,A -85,B 0,C 180,E1 -4236.083,E2 -4236.083} C_VEL
LIN {X 0,Y 530.586,Z 533.145,A -85,B 0,C 180,E1 -4237.229,E2 -4237.229} C_VEL
LIN {X 0,Y 530.776,Z 526.378,A -85,B 0,C 180,E1 -4238.566,E2 -4238.566} C_VEL
LIN {X 0,Y 530.921,Z 517.973,A -85,B 0,C 180,E1 -4239.909,E2 -4239.909} C_VEL
LIN {X 0,Y 531.221,Z 509.202,A -85,B 0,C 180,E1 -4241.06,E2 -4241.06} C_VEL
LIN {X 0,Y 531.497,Z 498.573,A -85,B 0,C 180,E1 -4242.214,E2 -4242.214} C_VEL
LIN {X 0,Y 531.814,Z 487.826,A -85,B 0,C 180,E1 -4243.177,E2 -4243.177} C_VEL
LIN {X 0,Y 532.192,Z 476.07,A -85,B 0,C 180,E1 -4244.043,E2 -4244.043} C_VEL
LIN {X 0,Y 532.557,Z 463.101,A -85,B 0,C 180,E1 -4244.814,E2 -4244.814} C_VEL
LIN {X 0,Y 532.905,Z 449.807,A -85,B 0,C 180,E1 -4245.428,E2 -4245.428} C_VEL
LIN {X 0,Y 533.122,Z 436.02,A -85,B 0,C 180,E1 -4245.901,E2 -4245.901} C_VEL
LIN {X 0,Y 533.287,Z 422.606,A -85,B 0,C 180,E1 -4246.213,E2 -4246.213} C_VEL
LIN {X 0,Y 533.939,Z 297.67,A -85,B 0,C 180,E1 -4247.93,E2 -4247.93} C_VEL
LIN {X 0,Y 531.863,Z 286.772,A -85,B 0,C 180,E1 -4248.174,E2 -4248.174} C_VEL
LIN {X 0,Y 532.036,Z 278.134,A -85,B 0,C 180,E1 -4249.483,E2 -4249.483} C_VEL
LIN {X 0,Y 532.502,Z 260.039,A -85,B 0,C 180,E1 -4252.35,E2 -4252.35} C_VEL
LIN {X 0,Y 531.066,Z 252.366,A -85,B 0,C 180,E1 -4253.667,E2 -4253.667} C_VEL
LIN {X 0,Y 530.967,Z 251.973,A -85,B 0,C 180,E1 -4253.95,E2 -4253.95} C_VEL
LIN {X 0,Y 531.005,Z 251.964,A -85,B 0,C 180,E1 -4256.743,E2 -4256.743} C_VEL
LIN {X 0,Y 530.981,Z 251.964,A -85,B 0,C 180,E1 -4259.322,E2 -4259.322} C_VEL
LIN {X 0,Y 530.969,Z 251.969,A -85,B 0,C 180,E1 -4262.1,E2 -4262.1} C_VEL
LIN {X 0,Y 530.981,Z 251.964,A -85,B 0,C 180,E1 -4264.852,E2 -4264.852} C_VEL
LIN {X 0,Y 530.964,Z 251.971,A -85,B 0,C 180,E1 -4267.507,E2 -4267.507} C_VEL
LIN {X 0,Y 530.981,Z 251.965,A -85,B 0,C 180,E1 -4270.432,E2 -4270.432} C_VEL
LIN {X 0,Y 530.967,Z 251.966,A -85,B 0,C 180,E1 -4273.281,E2 -4273.281} C_VEL
LIN {X 0,Y 530.984,Z 251.968,A -85,B 0,C 180,E1 -4275.62,E2 -4275.62} C_VEL
LIN {X 0,Y 531.001,Z 251.953,A -85,B 0,C 180,E1 -4278.565,E2 -4278.565} C_VEL
LIN {X 0,Y 530.963,Z 251.975,A -85,B 0,C 180,E1 -4281.345,E2 -4281.345} C_VEL
LIN {X 0,Y 530.976,Z 251.963,A -85,B 0,C 180,E1 -4284.381,E2 -4284.381} C_VEL
LIN {X 0,Y 530.966,Z 251.961,A -85,B 0,C 180,E1 -4287.133,E2 -4287.133} C_VEL
LIN {X 0,Y 530.979,Z 251.965,A -85,B 0,C 180,E1 -4289.804,E2 -4289.804} C_VEL
LIN {X 0,Y 531.009,Z 251.962,A -85,B 0,C 180,E1 -4292.466,E2 -4292.466} C_VEL
LIN {X 0,Y 530.998,Z 251.967,A -85,B 0,C 180,E1 -4294.942,E2 -4294.942} C_VEL
LIN {X 0,Y 530.963,Z 251.966,A -85,B 0,C 180,E1 -4298.246,E2 -4298.246} C_VEL
LIN {X 0,Y 530.989,Z 251.966,A -85,B 0,C 180,E1 -4300.677,E2 -4300.677} C_VEL
LIN {X 0,Y 530.985,Z 251.968,A -85,B 0,C 180,E1 -4303.071,E2 -4303.071} C_VEL
LIN {X 0,Y 531.01,Z 251.958,A -85,B 0,C 180,E1 -4305.436,E2 -4305.436} C_VEL
LIN {X 0,Y 531.038,Z 251.963,A -85,B 0,C 180,E1 -4308.55,E2 -4308.55} C_VEL
LIN {X 0,Y 531.048,Z 251.951,A -85,B 0,C 180,E1 -4311.629,E2 -4311.629} C_VEL
LIN {X 0,Y 531.131,Z 251.953,A -85,B 0,C 180,E1 -4314.685,E2 -4314.685} C_VEL
LIN {X 0,Y 531.13,Z 251.94,A -85,B 0,C 180,E1 -4317.725,E2 -4317.725} C_VEL
LIN {X 0,Y 531.147,Z 251.949,A -85,B 0,C 180,E1 -4320.758,E2 -4320.758} C_VEL
LIN {X 0,Y 531.1,Z 251.947,A -85,B 0,C 180,E1 -4323.034,E2 -4323.034} C_VEL
LIN {X 0,Y 531.076,Z 251.954,A -85,B 0,C 180,E1 -4326.077,E2 -4326.077} C_VEL
LIN {X 0,Y 531.027,Z 251.956,A -85,B 0,C 180,E1 -4329.138,E2 -4329.138} C_VEL
LIN {X 0,Y 531.032,Z 251.963,A -85,B 0,C 180,E1 -4332.225,E2 -4332.225} C_VEL
LIN {X 0,Y 530.987,Z 251.961,A -85,B 0,C 180,E1 -4335.35,E2 -4335.35} C_VEL
LIN {X 0,Y 531.008,Z 251.96,A -85,B 0,C 180,E1 -4337.723,E2 -4337.723} C_VEL
LIN {X 0,Y 530.991,Z 251.961,A -85,B 0,C 180,E1 -4340.938,E2 -4340.938} C_VEL
LIN {X 0,Y 530.972,Z 251.972,A -85,B 0,C 180,E1 -4344.225,E2 -4344.225} C_VEL
LIN {X 0,Y 530.998,Z 251.96,A -85,B 0,C 180,E1 -4346.744,E2 -4346.744} C_VEL
LIN {X 0,Y 530.993,Z 251.963,A -85,B 0,C 180,E1 -4349.322,E2 -4349.322} C_VEL
LIN {X 0,Y 530.973,Z 251.965,A -85,B 0,C 180,E1 -4352.104,E2 -4352.104} C_VEL
LIN {X 0,Y 530.982,Z 251.953,A -85,B 0,C 180,E1 -4354.855,E2 -4354.855} C_VEL
LIN {X 0,Y 530.96,Z 251.969,A -85,B 0,C 180,E1 -4357.508,E2 -4357.508} C_VEL
LIN {X 0,Y 530.979,Z 251.963,A -85,B 0,C 180,E1 -4360.433,E2 -4360.433} C_VEL
LIN {X 0,Y 530.958,Z 251.97,A -85,B 0,C 180,E1 -4363.282,E2 -4363.282} C_VEL
LIN {X 0,Y 530.984,Z 251.972,A -85,B 0,C 180,E1 -4365.621,E2 -4365.621} C_VEL
LIN {X 0,Y 531.004,Z 251.955,A -85,B 0,C 180,E1 -4368.567,E2 -4368.567} C_VEL
LIN {X 0,Y 530.965,Z 251.973,A -85,B 0,C 180,E1 -4371.347,E2 -4371.347} C_VEL
LIN {X 0,Y 530.952,Z 251.969,A -85,B 0,C 180,E1 -4374.381,E2 -4374.381} C_VEL
LIN {X 0,Y 530.969,Z 251.968,A -85,B 0,C 180,E1 -4377.134,E2 -4377.134} C_VEL
LIN {X 0,Y 530.968,Z 251.957,A -85,B 0,C 180,E1 -4379.804,E2 -4379.804} C_VEL
LIN {X 0,Y 531.014,Z 251.963,A -85,B 0,C 180,E1 -4382.468,E2 -4382.468} C_VEL
LIN {X 0,Y 531.063,Z 252.083,A -85,B 0,C 180,E1 -4385.208,E2 -4385.208} C_VEL
LIN {X 0,Y 532.704,Z 260.908,A -85,B 0,C 180,E1 -4386.685,E2 -4386.685} C_VEL
LIN {X 0,Y 532.134,Z 282.462,A -85,B 0,C 180,E1 -4389.917,E2 -4389.917} C_VEL
LIN {X 0,Y 531.841,Z 295.704,A -85,B 0,C 180,E1 -4391.853,E2 -4391.853} C_VEL
LIN {X 0,Y 533.053,Z 302.537,A -85,B 0,C 180,E1 -4392.02,E2 -4392.02} C_VEL
LIN {X 0,Y 533.908,Z 308.118,A -85,B 0,C 180,E1 -4392.126,E2 -4392.126} C_VEL
LIN {X 0,Y 533.274,Z 432.463,A -85,B 0,C 180,E1 -4393.835,E2 -4393.835} C_VEL
LIN {X 0,Y 533.05,Z 447.028,A -85,B 0,C 180,E1 -4394.183,E2 -4394.183} C_VEL
LIN {X 0,Y 532.772,Z 461.535,A -85,B 0,C 180,E1 -4394.703,E2 -4394.703} C_VEL
LIN {X 0,Y 532.458,Z 475.478,A -85,B 0,C 180,E1 -4395.379,E2 -4395.379} C_VEL
LIN {X 0,Y 532.047,Z 487.949,A -85,B 0,C 180,E1 -4396.148,E2 -4396.148} C_VEL
LIN {X 0,Y 531.693,Z 500.518,A -85,B 0,C 180,E1 -4397.112,E2 -4397.112} C_VEL
LIN {X 0,Y 531.417,Z 511.421,A -85,B 0,C 180,E1 -4398.14,E2 -4398.14} C_VEL
LIN {X 0,Y 531.114,Z 521.752,A -85,B 0,C 180,E1 -4399.324,E2 -4399.324} C_VEL
LIN {X 0,Y 530.9,Z 530.089,A -85,B 0,C 180,E1 -4400.476,E2 -4400.476} C_VEL
LIN {X 0,Y 530.709,Z 538.057,A -85,B 0,C 180,E1 -4401.816,E2 -4401.816} C_VEL
LIN {X 0,Y 530.572,Z 544.473,A -85,B 0,C 180,E1 -4403.153,E2 -4403.153} C_VEL
LIN {X 0,Y 530.514,Z 550.159,A -85,B 0,C 180,E1 -4404.679,E2 -4404.679} C_VEL
LIN {X 0,Y 530.497,Z 554.284,A -85,B 0,C 180,E1 -4406.202,E2 -4406.202} C_VEL
LIN {X 0,Y 530.41,Z 556.977,A -85,B 0,C 180,E1 -4407.722,E2 -4407.722} C_VEL
LIN {X 0,Y 530.341,Z 558.311,A -85,B 0,C 180,E1 -4409.241,E2 -4409.241} C_VEL
LIN {X 0,Y 530.341,Z 558.311,A -85,B 0,C 180,E1 -4410.759,E2 -4410.759} C_VEL
LIN {X 0,Y 530.41,Z 556.979,A -85,B 0,C 180,E1 -4412.278,E2 -4412.278} C_VEL
LIN {X 0,Y 530.497,Z 554.288,A -85,B 0,C 180,E1 -4413.798,E2 -4413.798} C_VEL
LIN {X 0,Y 530.514,Z 550.159,A -85,B 0,C 180,E1 -4415.321,E2 -4415.321} C_VEL
LIN {X 0,Y 530.572,Z 544.47,A -85,B 0,C 180,E1 -4416.847,E2 -4416.847} C_VEL
LIN {X 0,Y 530.709,Z 538.057,A -85,B 0,C 180,E1 -4418.184,E2 -4418.184} C_VEL
LIN {X 0,Y 530.899,Z 530.088,A -85,B 0,C 180,E1 -4419.525,E2 -4419.525} C_VEL
LIN {X 0,Y 531.114,Z 521.751,A -85,B 0,C 180,E1 -4420.676,E2 -4420.676} C_VEL
LIN {X 0,Y 531.454,Z 511.237,A -85,B 0,C 180,E1 -4421.879,E2 -4421.879} C_VEL
LIN {X 0,Y 531.719,Z 500.516,A -85,B 0,C 180,E1 -4422.888,E2 -4422.888} C_VEL
LIN {X 0,Y 532.078,Z 487.951,A -85,B 0,C 180,E1 -4423.851,E2 -4423.851} C_VEL
LIN {X 0,Y 532.472,Z 475.477,A -85,B 0,C 180,E1 -4424.621,E2 -4424.621} C_VEL
LIN {X 0,Y 532.761,Z 462.652,A -85,B 0,C 180,E1 -4425.248,E2 -4425.248} C_VEL
LIN {X 0,Y 533.035,Z 448.713,A -85,B 0,C 180,E1 -4425.763,E2 -4425.763} C_VEL
LIN {X 0,Y 533.268,Z 434.842,A -85,B 0,C 180,E1 -4426.116,E2 -4426.116} C_VEL
LIN {X 0,Y 533.447,Z 410.338,A -85,B 0,C 180,E1 -4426.479,E2 -4426.479} C_VEL
LIN {X 0,Y 533.849,Z 306.575,A -85,B 0,C 180,E1 -4427.897,E2 -4427.897} C_VEL
LIN {X 0,Y 531.873,Z 296.024,A -85,B 0,C 180,E1 -4428.125,E2 -4428.125} C_VEL
LIN {X 0,Y 531.931,Z 291.88,A -85,B 0,C 180,E1 -4428.687,E2 -4428.687} C_VEL
LIN {X 0,Y 532.356,Z 273.032,A -85,B 0,C 180,E1 -4431.49,E2 -4431.49} C_VEL
LIN {X 0,Y 532.708,Z 260.908,A -85,B 0,C 180,E1 -4433.315,E2 -4433.315} C_VEL
LIN {X 0,Y 531.063,Z 252.083,A -85,B 0,C 180,E1 -4434.793,E2 -4434.793} C_VEL
LIN {X 0,Y 531.015,Z 251.963,A -85,B 0,C 180,E1 -4437.595,E2 -4437.595} C_VEL
LIN {X 0,Y 530.973,Z 251.963,A -85,B 0,C 180,E1 -4440.645,E2 -4440.645} C_VEL
LIN {X 0,Y 530.985,Z 251.961,A -85,B 0,C 180,E1 -4443.772,E2 -4443.772} C_VEL
LIN {X 0,Y 530.952,Z 251.971,A -85,B 0,C 180,E1 -4446.558,E2 -4446.558} C_VEL
LIN {X 0,Y 530.982,Z 251.964,A -85,B 0,C 180,E1 -4449.443,E2 -4449.443} C_VEL
LIN {X 0,Y 530.979,Z 251.968,A -85,B 0,C 180,E1 -4452.456,E2 -4452.456} C_VEL
LIN {X 0,Y 530.981,Z 251.964,A -85,B 0,C 180,E1 -4455.62,E2 -4455.62} C_VEL
LIN {X 0,Y 530.995,Z 251.965,A -85,B 0,C 180,E1 -4458.564,E2 -4458.564} C_VEL
LIN {X 0,Y 530.954,Z 251.968,A -85,B 0,C 180,E1 -4461.529,E2 -4461.529} C_VEL
LIN {X 0,Y 530.976,Z 251.959,A -85,B 0,C 180,E1 -4464.382,E2 -4464.382} C_VEL
LIN {X 0,Y 530.966,Z 251.96,A -85,B 0,C 180,E1 -4467.133,E2 -4467.133} C_VEL
LIN {X 0,Y 530.98,Z 251.969,A -85,B 0,C 180,E1 -4469.804,E2 -4469.804} C_VEL
LIN {X 0,Y 531.011,Z 251.96,A -85,B 0,C 180,E1 -4472.466,E2 -4472.466} C_VEL
LIN {X 0,Y 531.001,Z 251.961,A -85,B 0,C 180,E1 -4474.942,E2 -4474.942} C_VEL
LIN {X 0,Y 530.963,Z 251.969,A -85,B 0,C 180,E1 -4478.246,E2 -4478.246} C_VEL
LIN {X 0,Y 530.989,Z 251.963,A -85,B 0,C 180,E1 -4480.677,E2 -4480.677} C_VEL
LIN {X 0,Y 530.985,Z 251.961,A -85,B 0,C 180,E1 -4483.071,E2 -4483.071} C_VEL
LIN {X 0,Y 531.011,Z 251.963,A -85,B 0,C 180,E1 -4485.436,E2 -4485.436} C_VEL
LIN {X 0,Y 531.028,Z 251.956,A -85,B 0,C 180,E1 -4488.55,E2 -4488.55} C_VEL
LIN {X 0,Y 531.049,Z 251.962,A -85,B 0,C 180,E1 -4491.629,E2 -4491.629} C_VEL
LIN {X 0,Y 531.115,Z 251.945,A -85,B 0,C 180,E1 -4494.685,E2 -4494.685} C_VEL
LIN {X 0,Y 531.131,Z 251.951,A -85,B 0,C 180,E1 -4497.725,E2 -4497.725} C_VEL
LIN {X 0,Y 531.147,Z 251.943,A -85,B 0,C 180,E1 -4500.758,E2 -4500.758} C_VEL
LIN {X 0,Y 531.101,Z 251.946,A -85,B 0,C 180,E1 -4503.034,E2 -4503.034} C_VEL
LIN {X 0,Y 531.076,Z 251.953,A -85,B 0,C 180,E1 -4506.077,E2 -4506.077} C_VEL
LIN {X 0,Y 531.025,Z 251.96,A -85,B 0,C 180,E1 -4509.138,E2 -4509.138} C_VEL
LIN {X 0,Y 531.033,Z 251.957,A -85,B 0,C 180,E1 -4512.225,E2 -4512.225} C_VEL
LIN {X 0,Y 530.988,Z 251.967,A -85,B 0,C 180,E1 -4515.35,E2 -4515.35} C_VEL
LIN {X 0,Y 531.009,Z 251.963,A -85,B 0,C 180,E1 -4517.723,E2 -4517.723} C_VEL
LIN {X 0,Y 530.992,Z 251.966,A -85,B 0,C 180,E1 -4520.938,E2 -4520.938} C_VEL
LIN {X 0,Y 530.973,Z 251.965,A -85,B 0,C 180,E1 -4524.225,E2 -4524.225} C_VEL
LIN {X 0,Y 531,Z 251.963,A -85,B 0,C 180,E1 -4526.744,E2 -4526.744} C_VEL
LIN {X 0,Y 530.994,Z 251.966,A -85,B 0,C 180,E1 -4529.322,E2 -4529.322} C_VEL
LIN {X 0,Y 530.974,Z 251.959,A -85,B 0,C 180,E1 -4532.104,E2 -4532.104} C_VEL
LIN {X 0,Y 530.984,Z 251.961,A -85,B 0,C 180,E1 -4534.855,E2 -4534.855} C_VEL
LIN {X 0,Y 530.962,Z 251.968,A -85,B 0,C 180,E1 -4537.508,E2 -4537.508} C_VEL
LIN {X 0,Y 530.996,Z 251.963,A -85,B 0,C 180,E1 -4540.432,E2 -4540.432} C_VEL
LIN {X 0,Y 530.961,Z 251.966,A -85,B 0,C 180,E1 -4543.495,E2 -4543.495} C_VEL
LIN {X 0,Y 530.958,Z 251.966,A -85,B 0,C 180,E1 -4543.572,E2 -4543.572} C_VEL
LIN {X 0,Y 530.286,Z 252.053,A -85,B 0,C 180,E1 -4544.206,E2 -4544.206} C_VEL
LIN {X 0,Y 527.44,Z 252.409,A -85,B 0,C 180,E1 -4545.235,E2 -4545.235} C_VEL
LIN {X 0,Y 525.038,Z 252.709,A -85,B 0,C 180,E1 -4546.063,E2 -4546.063} C_VEL
LIN {X 0,Y 524.005,Z 252.835,A -85,B 0,C 180,E1 -4546.703,E2 -4546.703} C_VEL
LIN {X 0,Y 523.92,Z 252.841,A -85,B 0,C 180,E1 -4546.92,E2 -4546.92} C_VEL
LIN {X 0,Y 523.946,Z 252.842,A -85,B 0,C 180,E1 -4549.921,E2 -4549.921} C_VEL
LIN {X 0,Y 523.909,Z 252.85,A -85,B 0,C 180,E1 -4552.869,E2 -4552.869} C_VEL
LIN {X 0,Y 523.94,Z 252.84,A -85,B 0,C 180,E1 -4555.711,E2 -4555.711} C_VEL
LIN {X 0,Y 523.923,Z 252.849,A -85,B 0,C 180,E1 -4558.457,E2 -4558.457} C_VEL
LIN {X 0,Y 523.939,Z 252.838,A -85,B 0,C 180,E1 -4561.126,E2 -4561.126} C_VEL
LIN {X 0,Y 523.985,Z 252.843,A -85,B 0,C 180,E1 -4563.981,E2 -4563.981} C_VEL
LIN {X 0,Y 523.95,Z 252.95,A -85,B 0,C 180,E1 -4566.131,E2 -4566.131} C_VEL
LIN {X 0,Y 525.365,Z 259.821,A -85,B 0,C 180,E1 -4567.375,E2 -4567.375} C_VEL
LIN {X 0,Y 525.523,Z 264.934,A -85,B 0,C 180,E1 -4568.216,E2 -4568.216} C_VEL
LIN {X 0,Y 524.905,Z 285.821,A -85,B 0,C 180,E1 -4571.548,E2 -4571.548} C_VEL
LIN {X 0,Y 525.002,Z 287.359,A -85,B 0,C 180,E1 -4571.692,E2 -4571.692} C_VEL
LIN {X 0,Y 527.187,Z 299.401,A -85,B 0,C 180,E1 -4571.946,E2 -4571.946} C_VEL
LIN {X 0,Y 526.49,Z 423.186,A -85,B 0,C 180,E1 -4573.671,E2 -4573.671} C_VEL
LIN {X 0,Y 526.223,Z 437.662,A -85,B 0,C 180,E1 -4574.024,E2 -4574.024} C_VEL
LIN {X 0,Y 525.993,Z 450.927,A -85,B 0,C 180,E1 -4574.501,E2 -4574.501} C_VEL
LIN {X 0,Y 525.708,Z 463.314,A -85,B 0,C 180,E1 -4575.088,E2 -4575.088} C_VEL
LIN {X 0,Y 525.259,Z 476.257,A -85,B 0,C 180,E1 -4575.867,E2 -4575.867} C_VEL
LIN {X 0,Y 524.904,Z 487.985,A -85,B 0,C 180,E1 -4576.745,E2 -4576.745} C_VEL
LIN {X 0,Y 524.496,Z 499.289,A -85,B 0,C 180,E1 -4577.777,E2 -4577.777} C_VEL
LIN {X 0,Y 524.223,Z 510.14,A -85,B 0,C 180,E1 -4578.987,E2 -4578.987} C_VEL
LIN {X 0,Y 523.899,Z 518.762,A -85,B 0,C 180,E1 -4580.152,E2 -4580.152} C_VEL
LIN {X 0,Y 523.693,Z 527.03,A -85,B 0,C 180,E1 -4581.511,E2 -4581.511} C_VEL
LIN {X 0,Y 523.54,Z 532.788,A -85,B 0,C 180,E1 -4582.673,E2 -4582.673} C_VEL
LIN {X 0,Y 523.469,Z 537.526,A -85,B 0,C 180,E1 -4583.834,E2 -4583.834} C_VEL
LIN {X 0,Y 523.376,Z 541.373,A -85,B 0,C 180,E1 -4584.993,E2 -4584.993} C_VEL
LIN {X 0,Y 523.419,Z 544.323,A -85,B 0,C 180,E1 -4586.151,E2 -4586.151} C_VEL
LIN {X 0,Y 523.334,Z 547.041,A -85,B 0,C 180,E1 -4587.691,E2 -4587.691} C_VEL
LIN {X 0,Y 523.246,Z 548.407,A -85,B 0,C 180,E1 -4589.23,E2 -4589.23} C_VEL
LIN {X 0,Y 523.247,Z 548.451,A -85,B 0,C 180,E1 -4590.77,E2 -4590.77} C_VEL
LIN {X 0,Y 523.333,Z 547.168,A -85,B 0,C 180,E1 -4592.309,E2 -4592.309} C_VEL
LIN {X 0,Y 523.419,Z 544.527,A -85,B 0,C 180,E1 -4593.849,E2 -4593.849} C_VEL
LIN {X 0,Y 523.451,Z 540.463,A -85,B 0,C 180,E1 -4595.393,E2 -4595.393} C_VEL
LIN {X 0,Y 523.497,Z 534.847,A -85,B 0,C 180,E1 -4596.94,E2 -4596.94} C_VEL
LIN {X 0,Y 523.665,Z 528.505,A -85,B 0,C 180,E1 -4598.295,E2 -4598.295} C_VEL
LIN {X 0,Y 523.883,Z 520.62,A -85,B 0,C 180,E1 -4599.653,E2 -4599.653} C_VEL
LIN {X 0,Y 524.115,Z 512.372,A -85,B 0,C 180,E1 -4600.82,E2 -4600.82} C_VEL
LIN {X 0,Y 524.432,Z 502.681,A -85,B 0,C 180,E1 -4601.961,E2 -4601.961} C_VEL
LIN {X 0,Y 524.763,Z 491.376,A -85,B 0,C 180,E1 -4603.061,E2 -4603.061} C_VEL
LIN {X 0,Y 525.115,Z 480.367,A -85,B 0,C 180,E1 -4603.94,E2 -4603.94} C_VEL
LIN {X 0,Y 525.549,Z 468.425,A -85,B 0,C 180,E1 -4604.719,E2 -4604.719} C_VEL
LIN {X 0,Y 525.889,Z 455.244,A -85,B 0,C 180,E1 -4605.403,E2 -4605.403} C_VEL
LIN {X 0,Y 526.206,Z 441.366,A -85,B 0,C 180,E1 -4605.946,E2 -4605.946} C_VEL
LIN {X 0,Y 526.437,Z 427.369,A -85,B 0,C 180,E1 -4606.331,E2 -4606.331} C_VEL
LIN {X 0,Y 526.613,Z 409.41,A -85,B 0,C 180,E1 -4606.624,E2 -4606.624} C_VEL
LIN {X 0,Y 527.084,Z 297.98,A -85,B 0,C 180,E1 -4608.167,E2 -4608.167} C_VEL
LIN {X 0,Y 524.965,Z 287.002,A -85,B 0,C 180,E1 -4608.413,E2 -4608.413} C_VEL
LIN {X 0,Y 524.928,Z 284.544,A -85,B 0,C 180,E1 -4608.743,E2 -4608.743} C_VEL
LIN {X 0,Y 525.545,Z 264.219,A -85,B 0,C 180,E1 -4611.989,E2 -4611.989} C_VEL
LIN {X 0,Y 525.455,Z 260.202,A -85,B 0,C 180,E1 -4612.649,E2 -4612.649} C_VEL
LIN {X 0,Y 523.96,Z 252.999,A -85,B 0,C 180,E1 -4613.938,E2 -4613.938} C_VEL
LIN {X 0,Y 523.975,Z 252.843,A -85,B 0,C 180,E1 -4616.271,E2 -4616.271} C_VEL
LIN {X 0,Y 523.953,Z 252.839,A -85,B 0,C 180,E1 -4619.323,E2 -4619.323} C_VEL
LIN {X 0,Y 523.935,Z 252.843,A -85,B 0,C 180,E1 -4622.449,E2 -4622.449} C_VEL
LIN {X 0,Y 523.93,Z 252.845,A -85,B 0,C 180,E1 -4625.225,E2 -4625.225} C_VEL
LIN {X 0,Y 523.913,Z 252.844,A -85,B 0,C 180,E1 -4628.101,E2 -4628.101} C_VEL
LIN {X 0,Y 523.959,Z 252.844,A -85,B 0,C 180,E1 -4631.31,E2 -4631.31} C_VEL
LIN {X 0,Y 523.952,Z 252.84,A -85,B 0,C 180,E1 -4634.691,E2 -4634.691} C_VEL
LIN {X 0,Y 523.951,Z 252.832,A -85,B 0,C 180,E1 -4637.881,E2 -4637.881} C_VEL
LIN {X 0,Y 523.973,Z 252.836,A -85,B 0,C 180,E1 -4639.923,E2 -4639.923} C_VEL
LIN {X 0,Y 523.906,Z 252.85,A -85,B 0,C 180,E1 -4642.868,E2 -4642.868} C_VEL
LIN {X 0,Y 523.938,Z 252.832,A -85,B 0,C 180,E1 -4645.71,E2 -4645.71} C_VEL
LIN {X 0,Y 523.926,Z 252.837,A -85,B 0,C 180,E1 -4648.456,E2 -4648.456} C_VEL
LIN {X 0,Y 523.945,Z 252.85,A -85,B 0,C 180,E1 -4651.125,E2 -4651.125} C_VEL
LIN {X 0,Y 523.976,Z 252.833,A -85,B 0,C 180,E1 -4653.98,E2 -4653.98} C_VEL
LIN {X 0,Y 523.928,Z 252.843,A -85,B 0,C 180,E1 -4656.27,E2 -4656.27} C_VEL
LIN {X 0,Y 523.938,Z 252.846,A -85,B 0,C 180,E1 -4658.766,E2 -4658.766} C_VEL
LIN {X 0,Y 523.945,Z 252.845,A -85,B 0,C 180,E1 -4661.22,E2 -4661.22} C_VEL
LIN {X 0,Y 523.932,Z 252.84,A -85,B 0,C 180,E1 -4663.639,E2 -4663.639} C_VEL
LIN {X 0,Y 523.932,Z 252.839,A -85,B 0,C 180,E1 -4666.028,E2 -4666.028} C_VEL
LIN {X 0,Y 524.003,Z 252.837,A -85,B 0,C 180,E1 -4668.394,E2 -4668.394} C_VEL
LIN {X 0,Y 523.997,Z 252.83,A -85,B 0,C 180,E1 -4671.516,E2 -4671.516} C_VEL
LIN {X 0,Y 524.09,Z 252.831,A -85,B 0,C 180,E1 -4674.614,E2 -4674.614} C_VEL
LIN {X 0,Y 524.103,Z 252.815,A -85,B 0,C 180,E1 -4677.694,E2 -4677.694} C_VEL
LIN {X 0,Y 524.117,Z 252.824,A -85,B 0,C 180,E1 -4680.768,E2 -4680.768} C_VEL
LIN {X 0,Y 524.067,Z 252.822,A -85,B 0,C 180,E1 -4683.075,E2 -4683.075} C_VEL
LIN {X 0,Y 524.038,Z 252.832,A -85,B 0,C 180,E1 -4686.159,E2 -4686.159} C_VEL
LIN {X 0,Y 523.994,Z 252.831,A -85,B 0,C 180,E1 -4689.262,E2 -4689.262} C_VEL
LIN {X 0,Y 523.993,Z 252.833,A -85,B 0,C 180,E1 -4691.74,E2 -4691.74} C_VEL
LIN {X 0,Y 523.983,Z 252.834,A -85,B 0,C 180,E1 -4695.053,E2 -4695.053} C_VEL
LIN {X 0,Y 523.955,Z 252.842,A -85,B 0,C 180,E1 -4697.969,E2 -4697.969} C_VEL
LIN {X 0,Y 523.963,Z 252.841,A -85,B 0,C 180,E1 -4700.41,E2 -4700.41} C_VEL
LIN {X 0,Y 523.908,Z 252.843,A -85,B 0,C 180,E1 -4702.894,E2 -4702.894} C_VEL
LIN {X 0,Y 523.944,Z 252.842,A -85,B 0,C 180,E1 -4705.419,E2 -4705.419} C_VEL
LIN {X 0,Y 523.962,Z 252.843,A -85,B 0,C 180,E1 -4707.999,E2 -4707.999} C_VEL
LIN {X 0,Y 523.945,Z 252.84,A -85,B 0,C 180,E1 -4710.857,E2 -4710.857} C_VEL
LIN {X 0,Y 523.954,Z 252.835,A -85,B 0,C 180,E1 -4713.735,E2 -4713.735} C_VEL
LIN {X 0,Y 523.916,Z 252.844,A -85,B 0,C 180,E1 -4716.405,E2 -4716.405} C_VEL
LIN {X 0,Y 523.918,Z 252.845,A -85,B 0,C 180,E1 -4719.085,E2 -4719.085} C_VEL
LIN {X 0,Y 523.951,Z 252.844,A -85,B 0,C 180,E1 -4722.119,E2 -4722.119} C_VEL
LIN {X 0,Y 523.951,Z 252.843,A -85,B 0,C 180,E1 -4725.309,E2 -4725.309} C_VEL
LIN {X 0,Y 523.969,Z 252.831,A -85,B 0,C 180,E1 -4728.688,E2 -4728.688} C_VEL
LIN {X 0,Y 523.921,Z 252.847,A -85,B 0,C 180,E1 -4731.08,E2 -4731.08} C_VEL
LIN {X 0,Y 523.898,Z 252.852,A -85,B 0,C 180,E1 -4733.826,E2 -4733.826} C_VEL
LIN {X 0,Y 523.94,Z 252.839,A -85,B 0,C 180,E1 -4736.636,E2 -4736.636} C_VEL
LIN {X 0,Y 523.954,Z 252.836,A -85,B 0,C 180,E1 -4739.356,E2 -4739.356} C_VEL
LIN {X 0,Y 523.977,Z 252.84,A -85,B 0,C 180,E1 -4742.282,E2 -4742.282} C_VEL
LIN {X 0,Y 524.02,Z 252.987,A -85,B 0,C 180,E1 -4745.01,E2 -4745.01} C_VEL
LIN {X 0,Y 525.8,Z 262.2,A -85,B 0,C 180,E1 -4746.569,E2 -4746.569} C_VEL
LIN {X 0,Y 525.253,Z 282.402,A -85,B 0,C 180,E1 -4749.642,E2 -4749.642} C_VEL
LIN {X 0,Y 524.923,Z 295.628,A -85,B 0,C 180,E1 -4751.605,E2 -4751.605} C_VEL
LIN {X 0,Y 526.089,Z 302.356,A -85,B 0,C 180,E1 -4751.772,E2 -4751.772} C_VEL
LIN {X 0,Y 527.155,Z 308.381,A -85,B 0,C 180,E1 -4751.894,E2 -4751.894} C_VEL
LIN {X 0,Y 526.461,Z 433.643,A -85,B 0,C 180,E1 -4753.645,E2 -4753.645} C_VEL
LIN {X 0,Y 526.2,Z 448.039,A -85,B 0,C 180,E1 -4754.007,E2 -4754.007} C_VEL
LIN {X 0,Y 525.881,Z 462.599,A -85,B 0,C 180,E1 -4754.547,E2 -4754.547} C_VEL
LIN {X 0,Y 525.582,Z 475.411,A -85,B 0,C 180,E1 -4755.183,E2 -4755.183} C_VEL
LIN {X 0,Y 525.14,Z 487.882,A -85,B 0,C 180,E1 -4755.962,E2 -4755.962} C_VEL
LIN {X 0,Y 524.722,Z 500.451,A -85,B 0,C 180,E1 -4756.937,E2 -4756.937} C_VEL
LIN {X 0,Y 524.452,Z 510.848,A -85,B 0,C 180,E1 -4757.926,E2 -4757.926} C_VEL
LIN {X 0,Y 524.097,Z 521.685,A -85,B 0,C 180,E1 -4759.18,E2 -4759.18} C_VEL
LIN {X 0,Y 523.854,Z 530.022,A -85,B 0,C 180,E1 -4760.346,E2 -4760.346} C_VEL
LIN {X 0,Y 523.634,Z 537.99,A -85,B 0,C 180,E1 -4761.705,E2 -4761.705} C_VEL
LIN {X 0,Y 523.494,Z 544.406,A -85,B 0,C 180,E1 -4763.06,E2 -4763.06} C_VEL
LIN {X 0,Y 523.448,Z 550.092,A -85,B 0,C 180,E1 -4764.607,E2 -4764.607} C_VEL
LIN {X 0,Y 523.419,Z 554.217,A -85,B 0,C 180,E1 -4766.151,E2 -4766.151} C_VEL
LIN {X 0,Y 523.333,Z 556.91,A -85,B 0,C 180,E1 -4767.691,E2 -4767.691} C_VEL
LIN {X 0,Y 523.247,Z 558.244,A -85,B 0,C 180,E1 -4769.23,E2 -4769.23} C_VEL
LIN {X 0,Y 523.247,Z 558.245,A -85,B 0,C 180,E1 -4770.77,E2 -4770.77} C_VEL
LIN {X 0,Y 523.333,Z 556.913,A -85,B 0,C 180,E1 -4772.309,E2 -4772.309} C_VEL
LIN {X 0,Y 523.419,Z 554.221,A -85,B 0,C 180,E1 -4773.849,E2 -4773.849} C_VEL
LIN {X 0,Y 523.449,Z 550.092,A -85,B 0,C 180,E1 -4775.393,E2 -4775.393} C_VEL
LIN {X 0,Y 523.494,Z 544.404,A -85,B 0,C 180,E1 -4776.94,E2 -4776.94} C_VEL
LIN {X 0,Y 523.635,Z 537.99,A -85,B 0,C 180,E1 -4778.296,E2 -4778.296} C_VEL
LIN {X 0,Y 523.853,Z 530.021,A -85,B 0,C 180,E1 -4779.654,E2 -4779.654} C_VEL
LIN {X 0,Y 524.098,Z 521.684,A -85,B 0,C 180,E1 -4780.82,E2 -4780.82} C_VEL
LIN {X 0,Y 524.448,Z 510.905,A -85,B 0,C 180,E1 -4782.068,E2 -4782.068} C_VEL
LIN {X 0,Y 524.75,Z 500.449,A -85,B 0,C 180,E1 -4783.062,E2 -4783.062} C_VEL
LIN {X 0,Y 525.159,Z 487.884,A -85,B 0,C 180,E1 -4784.037,E2 -4784.037} C_VEL
LIN {X 0,Y 525.58,Z 475.41,A -85,B 0,C 180,E1 -4784.817,E2 -4784.817} C_VEL
LIN {X 0,Y 525.921,Z 462.586,A -85,B 0,C 180,E1 -4785.452,E2 -4785.452} C_VEL
LIN {X 0,Y 526.197,Z 448.77,A -85,B 0,C 180,E1 -4785.969,E2 -4785.969} C_VEL
LIN {X 0,Y 526.466,Z 434.776,A -85,B 0,C 180,E1 -4786.33,E2 -4786.33} C_VEL
LIN {X 0,Y 526.644,Z 410.271,A -85,B 0,C 180,E1 -4786.698,E2 -4786.698} C_VEL
LIN {X 0,Y 527.059,Z 307.325,A -85,B 0,C 180,E1 -4788.124,E2 -4788.124} C_VEL
LIN {X 0,Y 524.935,Z 295.817,A -85,B 0,C 180,E1 -4788.382,E2 -4788.382} C_VEL
LIN {X 0,Y 525.438,Z 277.017,A -85,B 0,C 180,E1 -4791.17,E2 -4791.17} C_VEL
LIN {X 0,Y 525.797,Z 262.2,A -85,B 0,C 180,E1 -4793.431,E2 -4793.431} C_VEL
LIN {X 0,Y 524.02,Z 252.989,A -85,B 0,C 180,E1 -4794.99,E2 -4794.99} C_VEL
LIN {X 0,Y 523.969,Z 252.842,A -85,B 0,C 180,E1 -4797.998,E2 -4797.998} C_VEL
LIN {X 0,Y 523.943,Z 252.842,A -85,B 0,C 180,E1 -4800.854,E2 -4800.854} C_VEL
LIN {X 0,Y 523.957,Z 252.837,A -85,B 0,C 180,E1 -4803.734,E2 -4803.734} C_VEL
